C03578=1018.993,103.804,-130.711,-24.325,21.430,-41.754
C03579=1018.988,104.203,-130.749,-24.326,21.429,-41.751
C03580=1018.984,104.602,-130.786,-24.326,21.429,-41.747
C03581=1018.979,105.001,-130.824,-24.327,21.429,-41.743
C03582=1018.975,105.399,-130.861,-24.327,21.429,-41.740
C03583=1018.971,105.798,-130.899,-24.328,21.428,-41.736
C03584=1018.966,106.196,-130.936,-24.328,21.428,-41.734
C03585=1018.961,106.595,-130.974,-24.328,21.427,-41.730
C03586=1018.957,106.994,-131.011,-24.329,21.427,-41.727
C03587=1018.952,107.393,-131.049,-24.330,21.427,-41.723
C03588=1018.949,107.791,-131.087,-24.330,21.427,-41.719
C03589=1018.943,108.189,-131.124,-24.330,21.426,-41.717
C03590=1018.939,108.588,-131.162,-24.331,21.426,-41.714
C03591=1018.935,108.987,-131.199,-24.331,21.426,-41.710
C03592=1018.930,109.386,-131.237,-24.332,21.426,-41.707
C03593=1018.925,109.784,-131.275,-24.332,21.426,-41.703
C03594=1018.921,110.182,-131.312,-24.333,21.425,-41.701
C03595=1018.916,110.581,-131.350,-24.333,21.425,-41.697
C03596=1018.911,110.979,-131.388,-24.334,21.425,-41.694
C03597=1018.907,111.378,-131.425,-24.334,21.425,-41.690
C03598=1018.902,111.777,-131.463,-24.334,21.424,-41.688
C03599=1018.897,112.175,-131.500,-24.335,21.423,-41.684
C03600=1018.892,112.574,-131.539,-24.335,21.424,-41.681
C03601=1018.887,112.973,-131.577,-24.336,21.423,-41.677
C03602=1018.882,113.371,-131.613,-24.336,21.423,-41.675
C03603=1018.878,113.769,-131.652,-24.337,21.423,-41.671
C03604=1018.873,114.168,-131.689,-24.337,21.422,-41.668
C03605=1018.868,114.566,-131.727,-24.338,21.423,-41.664
C03606=1018.863,114.966,-131.765,-24.338,21.422,-41.662
C03607=1018.858,115.363,-131.803,-24.339,21.422,-41.659
C03608=1018.854,115.762,-131.840,-24.339,21.422,-41.655
C03609=1018.849,116.160,-131.878,-24.340,21.422,-41.652
C03610=1018.844,116.559,-131.916,-24.340,21.421,-41.649
C03611=1018.839,116.958,-131.953,-24.340,21.420,-41.646
C03612=1018.834,117.356,-131.991,-24.341,21.421,-41.642
C03613=1018.829,117.755,-132.029,-24.341,21.420,-41.638
C03614=1018.824,118.153,-132.067,-24.342,21.420,-41.637
C03615=1018.819,118.552,-132.105,-24.342,21.420,-41.633
C03616=1018.814,118.950,-132.143,-24.343,21.420,-41.629
C03617=1018.809,119.349,-132.180,-24.343,21.420,-41.626
C03618=1018.804,119.747,-132.218,-24.343,21.419,-41.624
C03619=1018.799,120.146,-132.256,-24.344,21.419,-41.620
C03620=1018.795,120.544,-132.294,-24.345,21.419,-41.617
C03621=1018.789,120.943,-132.332,-24.345,21.418,-41.614
C03622=1018.785,121.341,-132.370,-24.345,21.418,-41.611
C03623=1018.780,121.740,-132.408,-24.346,21.418,-41.607
C03624=1018.776,122.138,-132.447,-24.346,21.417,-41.605
C03625=1018.771,122.538,-132.484,-24.347,21.418,-41.602
C03626=1018.766,122.935,-132.522,-24.347,21.417,-41.598
C03627=1018.761,123.334,-132.561,-24.348,21.418,-41.595
C03628=1018.757,123.732,-132.599,-24.348,21.416,-41.592
C03629=1018.751,124.132,-132.637,-24.348,21.417,-41.589
C03630=1018.746,124.530,-132.675,-24.349,21.416,-41.585
C03631=1018.741,124.928,-132.714,-24.349,21.416,-41.583
C03632=1018.737,125.327,-132.751,-24.350,21.416,-41.580
C03633=1018.732,125.726,-132.790,-24.350,21.416,-41.576
C03634=1018.727,126.124,-132.828,-24.350,21.415,-41.574
C03635=1018.722,126.522,-132.867,-24.351,21.415,-41.571
C03636=1018.717,126.922,-132.904,-24.351,21.415,-41.567
C03637=1018.712,127.320,-132.943,-24.352,21.415,-41.565
C03638=1018.708,127.719,-132.981,-24.352,21.414,-41.561
C03639=1018.702,128.117,-133.019,-24.353,21.415,-41.558
C03640=1018.697,128.516,-133.057,-24.353,21.414,-41.555
C03641=1018.693,128.914,-133.096,-24.354,21.414,-41.552
C03642=1018.688,129.313,-133.134,-24.354,21.413,-41.550
C03643=1018.682,129.712,-133.172,-24.354,21.413,-41.547
C03644=1018.677,130.110,-133.210,-24.355,21.413,-41.543
C03645=1018.672,130.509,-133.249,-24.355,21.413,-41.541
C03646=1018.667,130.908,-133.287,-24.356,21.413,-41.538
C03647=1018.662,131.306,-133.325,-24.356,21.413,-41.534
C03648=1018.657,131.705,-133.364,-24.356,21.412,-41.532
C03649=1018.652,132.104,-133.402,-24.357,21.412,-41.528
C03650=1018.646,132.502,-133.440,-24.357,21.412,-41.525
C03651=1018.642,132.901,-133.479,-24.358,21.411,-41.523
C03652=1018.636,133.300,-133.517,-24.358,21.412,-41.519
C03653=1018.632,133.698,-133.555,-24.358,21.411,-41.517
C03654=1018.626,134.097,-133.594,-24.359,21.411,-41.514
C03655=1018.621,134.496,-133.632,-24.359,21.411,-41.510
C03656=1018.616,134.895,-133.671,-24.360,21.410,-41.508
C03657=1018.610,135.293,-133.710,-24.360,21.411,-41.505
C03658=1018.605,135.689,-133.747,-24.360,21.410,-41.502
C03659=1018.601,136.061,-133.783,-24.361,21.409,-41.500
C03660=1018.595,136.399,-133.815,-24.361,21.410,-41.497
C03661=1018.591,136.717,-133.846,-24.361,21.409,-41.495
C03662=1018.587,137.034,-133.876,-24.362,21.409,-41.491
C03663=1018.583,137.370,-133.909,-24.363,21.410,-41.488
C03664=1018.578,137.740,-133.944,-24.363,21.408,-41.486
C03665=1018.573,138.142,-133.983,-24.363,21.408,-41.484
C03666=1018.570,138.348,-134.003,-24.363,21.408,-41.482
C03667=1018.567,138.564,-134.024,-24.364,21.408,-41.480
C03668=1018.564,138.802,-134.047,-24.364,21.408,-41.478
C03669=1018.561,139.061,-134.072,-24.364,21.407,-41.476
C03670=1018.556,139.339,-134.099,-24.364,21.408,-41.475
C03671=1018.553,139.627,-134.126,-24.365,21.408,-41.473
C03672=1018.549,139.914,-134.154,-24.365,21.408,-41.471
C03673=1018.545,140.192,-134.182,-24.365,21.408,-41.470
C03674=1018.541,140.450,-134.206,-24.366,21.408,-41.468
C03675=1018.538,140.685,-134.229,-24.366,21.408,-41.466
C03676=1018.533,141.103,-134.269,-24.366,21.407,-41.462
C03677=1018.527,141.508,-134.308,-24.366,21.406,-41.460
C03678=1018.521,141.913,-134.347,-24.367,21.407,-41.457
C03679=1018.515,142.319,-134.386,-24.368,21.406,-41.453
C03680=1018.510,142.727,-134.425,-24.368,21.406,-41.451
C03681=1018.504,143.135,-134.466,-24.368,21.406,-41.448
C03682=1018.499,143.544,-134.505,-24.369,21.405,-41.445
C03683=1018.492,143.953,-134.544,-24.369,21.406,-41.442
C03684=1018.487,144.363,-134.584,-24.370,21.405,-41.438
C03685=1018.481,144.775,-134.624,-24.370,21.405,-41.436
C03686=1018.475,145.186,-134.664,-24.370,21.405,-41.432
C03687=1018.469,145.598,-134.704,-24.371,21.404,-41.431
C03688=1018.464,146.010,-134.743,-24.371,21.405,-41.427
C03689=1018.458,146.423,-134.783,-24.372,21.404,-41.424
C03690=1018.452,146.836,-134.823,-24.372,21.404,-41.422
C03691=1018.446,147.250,-134.863,-24.372,21.404,-41.418
C03692=1018.440,147.664,-134.904,-24.373,21.403,-41.416
C03693=1018.435,148.077,-134.943,-24.373,21.403,-41.412
C03694=1018.429,148.491,-134.983,-24.374,21.403,-41.409
C03695=1018.423,148.906,-135.023,-24.374,21.403,-41.407
C03696=1018.417,149.320,-135.064,-24.375,21.403,-41.403
C03697=1018.411,149.733,-135.103,-24.375,21.402,-41.401
C03698=1018.404,150.148,-135.144,-24.375,21.402,-41.398
C03699=1018.398,150.562,-135.184,-24.376,21.402,-41.394
C03700=1018.392,150.976,-135.224,-24.376,21.401,-41.392
C03701=1018.387,151.389,-135.264,-24.377,21.402,-41.389
C03702=1018.380,151.802,-135.304,-24.377,21.402,-41.387
C03703=1018.374,152.215,-135.345,-24.377,21.401,-41.383
C03704=1018.368,152.628,-135.384,-24.378,21.401,-41.381
C03705=1018.362,153.041,-135.424,-24.378,21.400,-41.377
C03706=1018.356,153.453,-135.465,-24.378,21.400,-41.375
C03707=1018.349,153.864,-135.504,-24.379,21.401,-41.372
C03708=1018.343,154.275,-135.544,-24.380,21.400,-41.368
C03709=1018.338,154.684,-135.584,-24.380,21.400,-41.366
C03710=1018.331,155.093,-135.624,-24.380,21.400,-41.363
C03711=1018.325,155.502,-135.663,-24.381,21.399,-41.361
C03712=1018.319,155.910,-135.703,-24.381,21.400,-41.358
C03713=1018.313,156.316,-135.742,-24.381,21.399,-41.355
C03714=1018.307,156.722,-135.782,-24.382,21.399,-41.352
C03715=1018.301,157.127,-135.821,-24.382,21.399,-41.350
C03716=1018.294,157.532,-135.861,-24.383,21.398,-41.346
C03717=1018.288,157.935,-135.899,-24.383,21.398,-41.344
C03718=1018.282,158.338,-135.939,-24.383,21.399,-41.341
C03719=1018.275,158.739,-135.978,-24.384,21.397,-41.339
C03720=1018.270,159.141,-136.017,-24.384,21.398,-41.335
C03721=1018.263,159.542,-136.055,-24.384,21.398,-41.333
C03722=1018.261,159.941,-136.098,-24.385,21.397,-41.330
C03723=1018.260,160.339,-136.139,-24.385,21.397,-41.328
C03724=1018.259,160.743,-136.182,-24.386,21.397,-41.325
C03725=1018.258,160.958,-136.203,-24.386,21.397,-41.324
C03726=1018.257,161.182,-136.227,-24.386,21.396,-41.322
C03727=1018.256,161.419,-136.252,-24.386,21.396,-41.320
C03728=1018.255,161.670,-136.279,-24.387,21.397,-41.319
C03729=1018.255,161.933,-136.307,-24.387,21.397,-41.317
C03730=1018.254,162.202,-136.334,-24.387,21.396,-41.315
C03731=1018.253,162.473,-136.362,-24.387,21.396,-41.313
C03732=1018.252,162.742,-136.392,-24.388,21.396,-41.311
C03733=1018.251,163.005,-136.419,-24.388,21.396,-41.309
C03734=1018.250,163.259,-136.445,-24.388,21.395,-41.308
C03735=1018.249,163.494,-136.470,-24.388,21.396,-41.306
C03736=1018.248,163.906,-136.513,-24.389,21.395,-41.304
C03737=1018.247,164.096,-136.533,-24.389,21.395,-41.302
C03738=1018.246,164.482,-136.574,-24.389,21.395,-41.300
C03739=1018.245,164.883,-136.616,-24.390,21.395,-41.297
C03740=1018.243,165.282,-136.658,-24.390,21.395,-41.295
C03741=1018.242,165.683,-136.700,-24.390,21.394,-41.291
C03742=1018.241,166.084,-136.743,-24.391,21.394,-41.289
C03743=1018.239,166.483,-136.785,-24.391,21.395,-41.286
C03744=1018.238,166.884,-136.827,-24.391,21.393,-41.284
C03745=1018.237,167.285,-136.870,-24.392,21.394,-41.280
C03746=1018.235,167.685,-136.911,-24.392,21.394,-41.278
C03747=1018.234,168.085,-136.954,-24.393,21.394,-41.275
C03748=1018.233,168.486,-136.996,-24.393,21.393,-41.273
C03749=1018.232,168.887,-137.039,-24.393,21.393,-41.271
C03750=1018.231,169.287,-137.081,-24.394,21.393,-41.267
C03751=1018.229,169.687,-137.123,-24.394,21.392,-41.265
C03752=1018.228,170.087,-137.165,-24.395,21.392,-41.262
C03753=1018.227,170.489,-137.208,-24.395,21.392,-41.260
C03754=1018.225,170.889,-137.250,-24.395,21.392,-41.256
C03755=1018.225,171.289,-137.293,-24.396,21.392,-41.254
C03756=1018.223,171.690,-137.335,-24.396,21.392,-41.251
C03757=1018.222,172.091,-137.378,-24.396,21.392,-41.249
C03758=1018.221,172.491,-137.420,-24.397,21.391,-41.247
C03759=1018.219,172.892,-137.463,-24.397,21.391,-41.243
C03760=1018.218,173.293,-137.506,-24.397,21.391,-41.242
C03761=1018.217,173.693,-137.548,-24.398,21.390,-41.238
C03762=1018.216,174.094,-137.590,-24.398,21.390,-41.236
C03763=1018.214,174.495,-137.633,-24.399,21.391,-41.233
C03764=1018.213,174.895,-137.676,-24.399,21.390,-41.231
C03765=1018.212,175.296,-137.718,-24.400,21.390,-41.227
C03766=1018.211,175.697,-137.761,-24.400,21.390,-41.225
C03767=1018.210,176.098,-137.804,-24.400,21.390,-41.223
C03768=1018.209,176.498,-137.847,-24.401,21.389,-41.219
C03769=1018.207,176.899,-137.889,-24.401,21.389,-41.218
C03770=1018.206,177.299,-137.931,-24.401,21.389,-41.214
C03771=1018.206,177.701,-137.975,-24.402,21.389,-41.212
C03772=1018.204,178.101,-138.018,-24.402,21.389,-41.209
C03773=1018.203,178.502,-138.060,-24.402,21.388,-41.207
C03774=1018.202,178.904,-138.103,-24.403,21.388,-41.205
C03775=1018.201,179.304,-138.146,-24.403,21.388,-41.201
C03776=1018.200,179.704,-138.189,-24.403,21.388,-41.199
C03777=1018.199,180.105,-138.232,-24.404,21.388,-41.196
C03778=1018.198,180.506,-138.275,-24.404,21.388,-41.194
C03779=1018.197,180.908,-138.317,-24.405,21.387,-41.190
C03780=1018.195,181.308,-138.360,-24.405,21.387,-41.188
C03781=1018.194,181.709,-138.403,-24.405,21.387,-41.186
C03782=1018.193,182.110,-138.447,-24.406,21.387,-41.183
C03783=1018.192,182.511,-138.490,-24.406,21.386,-41.181
C03784=1018.191,182.912,-138.533,-24.407,21.387,-41.177
C03785=1018.190,183.312,-138.576,-24.407,21.386,-41.176
C03786=1018.189,183.713,-138.619,-24.407,21.386,-41.172
C03787=1018.188,184.115,-138.662,-24.408,21.386,-41.170
C03788=1018.187,184.515,-138.705,-24.408,21.386,-41.168
C03789=1018.186,184.917,-138.748,-24.409,21.386,-41.165
C03790=1018.185,185.318,-138.791,-24.409,21.385,-41.162
C03791=1018.184,185.719,-138.834,-24.409,21.385,-41.159
C03792=1018.183,186.120,-138.878,-24.410,21.385,-41.157
C03793=1018.182,186.521,-138.921,-24.410,21.384,-41.155
C03794=1018.181,186.922,-138.964,-24.410,21.384,-41.151
C03795=1018.180,187.323,-139.007,-24.411,21.384,-41.150
C03796=1018.180,187.723,-139.051,-24.411,21.385,-41.146
C03797=1018.179,188.125,-139.095,-24.411,21.384,-41.144
C03798=1018.178,188.525,-139.137,-24.412,21.384,-41.141
C03799=1018.177,188.926,-139.181,-24.412,21.384,-41.139
C03800=1018.176,189.328,-139.224,-24.412,21.384,-41.137
C03801=1018.176,189.729,-139.267,-24.413,21.383,-41.133
C03802=1018.175,190.130,-139.311,-24.413,21.383,-41.131
C03803=1018.174,190.531,-139.354,-24.414,21.383,-41.128
C03804=1018.173,190.932,-139.397,-24.414,21.383,-41.126
C03805=1018.172,191.333,-139.442,-24.414,21.382,-41.124
C03806=1018.171,191.734,-139.485,-24.415,21.382,-41.120
C03807=1018.170,192.135,-139.528,-24.415,21.382,-41.118
C03808=1018.169,192.536,-139.572,-24.415,21.382,-41.115
C03809=1018.169,192.938,-139.615,-24.416,21.382,-41.113
C03810=1018.168,193.338,-139.659,-24.416,21.382,-41.109
C03811=1018.167,193.739,-139.702,-24.417,21.382,-41.108
C03812=1018.166,194.141,-139.746,-24.417,21.381,-41.105
C03813=1018.165,194.541,-139.790,-24.417,21.381,-41.102
C03814=1018.165,194.943,-139.833,-24.418,21.381,-41.100
C03815=1018.164,195.345,-139.877,-24.418,21.381,-41.097
C03816=1018.164,195.745,-139.921,-24.418,21.380,-41.094
C03817=1018.163,196.147,-139.965,-24.419,21.381,-41.091
C03818=1018.162,196.548,-140.008,-24.419,21.380,-41.089
C03819=1018.161,196.949,-140.052,-24.419,21.380,-41.087
C03820=1018.161,197.350,-140.096,-24.420,21.380,-41.084
C03821=1018.160,197.750,-140.140,-24.420,21.380,-41.082
C03822=1018.159,198.153,-140.184,-24.421,21.380,-41.078
C03823=1018.159,198.554,-140.227,-24.421,21.379,-41.076
C03824=1018.158,198.954,-140.271,-24.421,21.379,-41.074
C03825=1018.158,199.353,-140.315,-24.422,21.379,-41.071
C03826=1018.157,199.742,-140.358,-24.422,21.379,-41.069
C03827=1018.156,200.142,-140.401,-24.423,21.378,-41.065
C03828=1018.156,200.355,-140.425,-24.423,21.378,-41.065
C03829=1018.156,200.577,-140.449,-24.423,21.378,-41.063
C03830=1018.156,200.807,-140.475,-24.423,21.378,-41.061
C03831=1018.155,201.034,-140.500,-24.423,21.379,-41.060
C03832=1018.154,201.442,-140.544,-24.424,21.378,-41.058
C03833=1018.154,201.793,-140.582,-24.424,21.378,-41.054
C03834=1018.155,202.143,-140.622,-24.424,21.378,-41.052
C03835=1018.156,202.530,-140.666,-24.425,21.378,-41.051
C03836=1018.162,203.746,-140.801,-24.373,21.403,-41.416
C03837=1018.164,203.994,-140.828,-24.373,21.404,-41.415
C03838=1018.166,204.242,-140.857,-24.373,21.403,-41.414
C03839=1018.168,204.491,-140.884,-24.373,21.403,-41.412
C03840=1018.170,204.739,-140.911,-24.374,21.404,-41.411
C03841=1018.172,204.988,-140.939,-24.373,21.403,-41.410
C03842=1018.174,205.237,-140.966,-24.374,21.403,-41.409
C03843=1018.176,205.486,-140.994,-24.374,21.403,-41.407
C03844=1018.178,205.734,-141.021,-24.374,21.402,-41.407
C03845=1018.180,205.982,-141.049,-24.374,21.403,-41.405
C03846=1018.181,206.231,-141.076,-24.375,21.403,-41.403
C03847=1018.184,206.479,-141.104,-24.375,21.402,-41.401
C03848=1018.186,206.727,-141.131,-24.375,21.402,-41.401
C03849=1018.187,206.976,-141.158,-24.375,21.402,-41.399
C03850=1018.189,207.224,-141.186,-24.375,21.402,-41.398
C03851=1018.192,207.473,-141.213,-24.375,21.402,-41.398
C03852=1018.193,207.722,-141.241,-24.376,21.402,-41.396
C03853=1018.196,207.970,-141.269,-24.376,21.402,-41.394
C03854=1018.198,208.218,-141.296,-24.376,21.402,-41.392
C03855=1018.199,208.461,-141.323,-24.376,21.401,-41.392
C03856=1018.201,208.704,-141.350,-24.376,21.402,-41.391
C03857=1018.203,208.946,-141.377,-24.377,21.402,-41.389
C03858=1018.206,209.189,-141.404,-24.377,21.401,-41.388
C03859=1018.208,209.432,-141.430,-24.377,21.402,-41.387
C03860=1018.209,209.675,-141.458,-24.377,21.401,-41.385
C03861=1018.212,209.917,-141.485,-24.377,21.401,-41.383
C03862=1018.213,210.160,-141.512,-24.377,21.401,-41.383
C03863=1018.216,210.408,-141.540,-24.378,21.401,-41.381
C03864=1018.217,210.657,-141.567,-24.378,21.401,-41.379
C03865=1018.220,210.905,-141.595,-24.378,21.401,-41.378
C03866=1018.222,211.153,-141.622,-24.378,21.400,-41.377
C03867=1018.224,211.402,-141.651,-24.378,21.400,-41.375
C03868=1018.226,211.651,-141.677,-24.379,21.401,-41.374
C03869=1018.228,211.899,-141.706,-24.379,21.401,-41.372
C03870=1018.230,212.148,-141.733,-24.379,21.400,-41.372
C03871=1018.233,212.396,-141.761,-24.379,21.400,-41.370
C03872=1018.234,212.644,-141.789,-24.380,21.400,-41.368
C03873=1018.236,212.893,-141.816,-24.380,21.400,-41.366
C03874=1018.239,213.141,-141.844,-24.380,21.400,-41.366
C03875=1018.241,213.460,-141.879,-24.380,21.400,-41.365
C03876=1018.244,213.778,-141.915,-24.380,21.400,-41.363
C03877=1018.247,214.097,-141.951,-24.381,21.399,-41.361
C03878=1018.250,214.416,-141.986,-24.381,21.399,-41.359
C03879=1018.252,214.665,-142.015,-24.381,21.399,-41.357
C03880=1018.254,214.912,-142.042,-24.381,21.400,-41.356
C03881=1018.256,215.160,-142.070,-24.382,21.399,-41.354
C03882=1018.258,215.410,-142.098,-24.382,21.399,-41.352
C03883=1018.262,215.825,-142.145,-24.382,21.399,-41.350
C03884=1018.266,216.240,-142.191,-24.382,21.399,-41.348
C03885=1018.270,216.656,-142.237,-24.383,21.399,-41.345
C03886=1018.274,217.071,-142.284,-24.383,21.398,-41.342
C03887=1018.276,217.319,-142.311,-24.383,21.399,-41.341
C03888=1018.278,217.568,-142.340,-24.384,21.398,-41.339
C03889=1018.281,217.816,-142.368,-24.384,21.397,-41.339
C03890=1018.282,218.065,-142.395,-24.384,21.397,-41.337
C03891=1018.285,218.314,-142.423,-24.384,21.398,-41.335
C03892=1018.287,218.561,-142.451,-24.384,21.398,-41.333
C03893=1018.289,218.810,-142.480,-24.385,21.397,-41.332
C03894=1018.292,219.058,-142.508,-24.385,21.397,-41.330
C03895=1018.294,219.307,-142.535,-24.385,21.397,-41.330
C03896=1018.296,219.556,-142.563,-24.385,21.397,-41.328
C03897=1018.298,219.804,-142.591,-24.385,21.397,-41.326
C03898=1018.301,220.052,-142.619,-24.386,21.397,-41.324
C03899=1018.303,220.300,-142.647,-24.386,21.397,-41.323
C03900=1018.306,220.549,-142.675,-24.386,21.397,-41.321
C03901=1018.308,220.797,-142.703,-24.386,21.396,-41.320
C03902=1018.311,221.046,-142.732,-24.386,21.396,-41.318
C03903=1018.313,221.294,-142.759,-24.387,21.397,-41.317
C03904=1018.316,221.542,-142.787,-24.387,21.396,-41.315
C03905=1018.318,221.791,-142.816,-24.387,21.396,-41.313
C03906=1018.320,222.040,-142.843,-24.388,21.396,-41.311
C03907=1018.322,222.282,-142.870,-24.388,21.397,-41.310
C03908=1018.325,222.526,-142.898,-24.388,21.396,-41.309
C03909=1018.327,222.768,-142.926,-24.388,21.395,-41.308
C03910=1018.330,223.011,-142.953,-24.388,21.395,-41.306
C03911=1018.332,223.254,-142.981,-24.389,21.396,-41.304
C03912=1018.334,223.497,-143.008,-24.389,21.396,-41.302
C03913=1018.337,223.740,-143.036,-24.389,21.395,-41.300
C03914=1018.339,223.983,-143.063,-24.389,21.395,-41.300
C03915=1018.342,224.231,-143.092,-24.389,21.394,-41.298
C03916=1018.344,224.479,-143.119,-24.390,21.395,-41.297
C03917=1018.346,224.728,-143.148,-24.390,21.395,-41.295
C03918=1018.349,224.976,-143.177,-24.390,21.395,-41.293
C03919=1018.352,225.224,-143.204,-24.390,21.394,-41.291
C03920=1018.354,225.473,-143.233,-24.391,21.394,-41.289
C03921=1018.356,225.721,-143.261,-24.391,21.395,-41.288
C03922=1018.359,225.969,-143.289,-24.391,21.395,-41.286
C03923=1018.361,226.218,-143.317,-24.391,21.394,-41.285
C03924=1018.364,226.466,-143.345,-24.391,21.393,-41.284
C03925=1018.366,226.715,-143.374,-24.392,21.393,-41.282
C03926=1018.369,226.964,-143.402,-24.392,21.394,-41.280
C03927=1018.372,227.211,-143.430,-24.392,21.394,-41.278
C03928=1018.374,227.460,-143.459,-24.393,21.393,-41.276
C03929=1018.377,227.709,-143.487,-24.393,21.393,-41.275
C03930=1018.379,227.956,-143.515,-24.393,21.393,-41.273
C03931=1018.381,228.205,-143.543,-24.393,21.394,-41.271
C03932=1018.384,228.454,-143.571,-24.394,21.393,-41.269
C03933=1018.388,228.702,-143.600,-24.394,21.393,-41.267
C03934=1018.389,228.950,-143.629,-24.394,21.393,-41.266
C03935=1018.392,229.193,-143.656,-24.394,21.392,-41.265
C03936=1018.395,229.437,-143.684,-24.394,21.392,-41.263
C03937=1018.397,229.679,-143.711,-24.395,21.392,-41.262
C03938=1018.400,229.922,-143.740,-24.395,21.392,-41.260
C03939=1018.403,230.165,-143.767,-24.395,21.392,-41.258
C03940=1018.405,230.408,-143.795,-24.395,21.392,-41.256
C03941=1018.408,230.651,-143.823,-24.396,21.392,-41.254
C03942=1018.410,230.895,-143.851,-24.396,21.391,-41.252
C03943=1018.413,231.143,-143.880,-24.396,21.392,-41.251
C03944=1018.416,231.391,-143.907,-24.396,21.392,-41.249
C03945=1018.418,231.640,-143.936,-24.397,21.392,-41.247
C03946=1018.421,231.888,-143.965,-24.397,21.391,-41.245
C03947=1018.424,232.136,-143.993,-24.397,21.391,-41.243
C03948=1018.426,232.384,-144.022,-24.397,21.391,-41.242
C03949=1018.429,232.633,-144.050,-24.398,21.391,-41.240
C03950=1018.432,232.881,-144.078,-24.398,21.390,-41.238
C03951=1018.434,233.129,-144.107,-24.398,21.391,-41.236
C03952=1018.437,233.378,-144.135,-24.399,21.391,-41.234
C03953=1018.440,233.626,-144.165,-24.399,21.391,-41.233
C03954=1018.443,233.875,-144.193,-24.399,21.390,-41.231
C03955=1018.446,234.123,-144.221,-24.399,21.390,-41.229
C03956=1018.448,234.372,-144.250,-24.400,21.390,-41.227
C03957=1018.451,234.620,-144.278,-24.400,21.390,-41.225
C03958=1018.453,234.868,-144.307,-24.400,21.390,-41.223
C03959=1018.456,235.116,-144.335,-24.400,21.389,-41.221
C03960=1018.459,235.364,-144.364,-24.401,21.389,-41.219
C03961=1018.462,235.613,-144.393,-24.401,21.389,-41.218
C03962=1018.465,235.861,-144.422,-24.401,21.390,-41.216
C03963=1018.468,236.104,-144.449,-24.401,21.389,-41.214
C03964=1018.470,236.347,-144.478,-24.402,21.389,-41.212
C03965=1018.473,236.590,-144.506,-24.402,21.389,-41.210
C03966=1018.476,236.834,-144.534,-24.402,21.389,-41.209
C03967=1018.479,237.077,-144.562,-24.402,21.388,-41.207
C03968=1018.481,237.320,-144.590,-24.403,21.388,-41.205
C03969=1018.484,237.563,-144.618,-24.403,21.388,-41.203
C03970=1018.487,237.806,-144.646,-24.403,21.388,-41.201
C03971=1018.490,238.054,-144.675,-24.403,21.388,-41.199
C03972=1018.493,238.303,-144.703,-24.404,21.387,-41.197
C03973=1018.495,238.551,-144.733,-24.404,21.387,-41.195
C03974=1018.499,238.799,-144.762,-24.405,21.388,-41.192
C03975=1018.501,239.048,-144.790,-24.405,21.387,-41.190
C03976=1018.504,239.296,-144.819,-24.405,21.387,-41.188
C03977=1018.507,239.544,-144.848,-24.405,21.387,-41.186
C03978=1018.510,239.793,-144.876,-24.406,21.387,-41.184
C03979=1018.513,240.041,-144.905,-24.406,21.386,-41.183
C03980=1018.517,240.290,-144.934,-24.406,21.386,-41.181
C03981=1018.519,240.538,-144.964,-24.406,21.386,-41.179
C03982=1018.522,240.786,-144.992,-24.407,21.386,-41.177
C03983=1018.525,241.034,-145.021,-24.407,21.386,-41.174
C03984=1018.528,241.283,-145.050,-24.407,21.386,-41.172
C03985=1018.531,241.531,-145.079,-24.408,21.386,-41.170
C03986=1018.533,241.780,-145.107,-24.408,21.386,-41.168
C03987=1018.537,242.028,-145.136,-24.408,21.385,-41.166
C03988=1018.540,242.275,-145.165,-24.408,21.385,-41.164
C03989=1018.543,242.524,-145.195,-24.409,21.385,-41.162
C03990=1018.546,242.772,-145.224,-24.409,21.385,-41.159
C03991=1018.549,243.016,-145.252,-24.410,21.385,-41.157
C03992=1018.552,243.259,-145.280,-24.410,21.385,-41.155
C03993=1018.555,243.502,-145.309,-24.410,21.385,-41.153
C03994=1018.558,243.745,-145.337,-24.410,21.384,-41.151
C03995=1018.560,243.988,-145.366,-24.411,21.384,-41.150
C03996=1018.564,244.232,-145.394,-24.411,21.384,-41.148
C03997=1018.567,244.475,-145.422,-24.411,21.384,-41.144
C03998=1018.570,244.718,-145.451,-24.412,21.384,-41.143
C03999=1018.573,244.967,-145.480,-24.412,21.384,-41.141
C04000=1018.576,245.215,-145.509,-24.412,21.384,-41.139
C04001=1018.579,245.463,-145.538,-24.412,21.384,-41.137
C04002=1018.582,245.711,-145.567,-24.413,21.384,-41.134
C04003=1018.586,245.960,-145.596,-24.413,21.384,-41.132
C04004=1018.588,246.208,-145.626,-24.413,21.383,-41.129
C04005=1018.592,246.456,-145.655,-24.414,21.382,-41.127
C04006=1018.595,246.704,-145.683,-24.414,21.382,-41.126
C04007=1018.598,246.953,-145.713,-24.414,21.383,-41.122
C04008=1018.601,247.201,-145.742,-24.415,21.382,-41.120
C04009=1018.604,247.449,-145.771,-24.415,21.382,-41.118
C04010=1018.607,247.697,-145.800,-24.415,21.382,-41.117
C04011=1018.610,247.946,-145.830,-24.416,21.382,-41.113
C04012=1018.613,248.194,-145.859,-24.416,21.382,-41.111
C04013=1018.617,248.443,-145.888,-24.416,21.381,-41.109
C04014=1018.620,248.690,-145.918,-24.417,21.381,-41.107
C04015=1018.623,248.938,-145.947,-24.417,21.381,-41.104
C04016=1018.627,249.187,-145.976,-24.417,21.381,-41.102
C04017=1018.630,249.435,-146.005,-24.418,21.381,-41.100
C04018=1018.632,249.684,-146.035,-24.418,21.381,-41.098
C04019=1018.636,249.927,-146.063,-24.418,21.381,-41.095
C04020=1018.639,250.171,-146.092,-24.419,21.381,-41.093
C04021=1018.643,250.413,-146.121,-24.419,21.380,-41.091
C04022=1018.646,250.657,-146.150,-24.419,21.380,-41.089
C04023=1018.649,250.901,-146.178,-24.420,21.380,-41.085
C04024=1018.652,251.144,-146.207,-24.420,21.380,-41.084
C04025=1018.655,251.387,-146.236,-24.420,21.380,-41.082
C04026=1018.659,251.631,-146.265,-24.421,21.380,-41.078
C04027=1018.661,251.879,-146.294,-24.421,21.380,-41.076
C04028=1018.666,252.127,-146.324,-24.421,21.379,-41.074
C04029=1018.668,252.375,-146.353,-24.421,21.378,-41.072
C04030=1018.671,252.623,-146.382,-24.422,21.379,-41.069
C04031=1018.675,252.872,-146.412,-24.422,21.379,-41.067
C04032=1018.678,253.120,-146.441,-24.423,21.378,-41.065
C04033=1018.681,253.369,-146.471,-24.423,21.378,-41.061
C04034=1018.685,253.616,-146.500,-24.423,21.378,-41.060
C04035=1018.689,253.865,-146.530,-24.424,21.378,-41.058
C04036=1018.691,254.112,-146.560,-24.424,21.378,-41.054
C04037=1018.695,254.361,-146.589,-24.424,21.378,-41.052
C04038=1018.698,254.609,-146.618,-24.425,21.377,-41.049
C04039=1018.702,254.857,-146.648,-24.425,21.377,-41.047
C04040=1018.705,255.106,-146.678,-24.425,21.377,-41.045
C04041=1018.709,255.354,-146.707,-24.426,21.377,-41.042
C04042=1018.712,255.603,-146.737,-24.426,21.377,-41.040
C04043=1018.715,255.850,-146.767,-24.426,21.376,-41.037
C04044=1018.718,256.099,-146.796,-24.427,21.376,-41.034
C04045=1018.723,256.347,-146.826,-24.427,21.376,-41.032
C04046=1018.725,256.595,-146.856,-24.428,21.377,-41.029
C04047=1018.729,256.839,-146.884,-24.428,21.376,-41.027
C04048=1018.732,257.082,-146.913,-24.428,21.375,-41.025
C04049=1018.735,257.326,-146.943,-24.429,21.376,-41.021
C04050=1018.739,257.568,-146.972,-24.429,21.376,-41.019
C04051=1018.743,257.812,-147.001,-24.429,21.375,-41.018
C04052=1018.746,258.056,-147.030,-24.430,21.375,-41.014
C04053=1018.750,258.299,-147.059,-24.430,21.375,-41.012
C04054=1018.767,259.535,-147.213,-24.551,21.322,-40.171
C04055=1018.770,259.815,-147.250,-24.587,21.310,-39.930
C04056=1018.772,260.095,-147.287,-24.622,21.298,-39.688
C04057=1018.774,260.374,-147.326,-24.658,21.287,-39.446
C04058=1018.775,260.654,-147.364,-24.693,21.275,-39.204
C04059=1018.776,260.901,-147.398,-24.725,21.267,-38.988
C04060=1018.776,261.149,-147.433,-24.758,21.259,-38.770
C04061=1018.776,261.396,-147.469,-24.790,21.251,-38.554
C04062=1018.776,261.644,-147.505,-24.823,21.245,-38.337
C04063=1018.776,261.924,-147.546,-24.860,21.238,-38.090
C04064=1018.775,262.203,-147.589,-24.897,21.233,-37.842
C04065=1018.773,262.482,-147.632,-24.935,21.227,-37.593
C04066=1018.770,262.761,-147.675,-24.973,21.223,-37.345
C04067=1018.769,263.008,-147.713,-25.006,21.220,-37.124
C04068=1018.767,263.255,-147.753,-25.040,21.217,-36.903
C04069=1018.764,263.502,-147.793,-25.074,21.216,-36.681
C04070=1018.760,263.749,-147.833,-25.108,21.215,-36.458
C04071=1018.755,264.028,-147.880,-25.147,21.216,-36.205
C04072=1018.752,264.307,-147.928,-25.186,21.217,-35.952
C04073=1018.747,264.586,-147.975,-25.226,21.219,-35.699
C04074=1018.741,264.865,-148.023,-25.265,21.221,-35.444
C04075=1018.736,265.112,-148.067,-25.300,21.225,-35.219
C04076=1018.730,265.358,-148.111,-25.335,21.229,-34.991
C04077=1018.724,265.604,-148.154,-25.370,21.233,-34.766
C04078=1018.718,265.850,-148.199,-25.406,21.239,-34.538
C04079=1018.710,266.128,-148.251,-25.446,21.246,-34.279
C04080=1018.702,266.408,-148.303,-25.487,21.254,-34.021
C04081=1018.693,266.686,-148.356,-25.527,21.264,-33.760
C04082=1018.684,266.965,-148.409,-25.568,21.275,-33.499
C04083=1018.677,267.210,-148.457,-25.604,21.284,-33.269
C04084=1018.667,267.455,-148.505,-25.641,21.295,-33.037
C04085=1018.658,267.701,-148.554,-25.677,21.306,-32.805
C04086=1018.649,267.946,-148.604,-25.714,21.319,-32.571
C04087=1018.638,268.224,-148.659,-25.755,21.333,-32.307
C04088=1018.627,268.503,-148.717,-25.797,21.350,-32.039
C04089=1018.614,268.782,-148.775,-25.839,21.367,-31.772
C04090=1018.601,269.060,-148.833,-25.881,21.386,-31.502
C04091=1018.590,269.304,-148.885,-25.918,21.402,-31.266
C04092=1018.578,269.549,-148.937,-25.955,21.420,-31.029
C04093=1018.566,269.792,-148.991,-25.992,21.439,-30.791
C04094=1018.554,270.037,-149.045,-26.030,21.459,-30.551
C04095=1018.539,270.315,-149.107,-26.072,21.483,-30.277
C04096=1018.524,270.594,-149.169,-26.115,21.507,-30.003
C04097=1018.508,270.871,-149.232,-26.158,21.533,-29.728
C04098=1018.491,271.150,-149.296,-26.201,21.560,-29.450
C04099=1018.477,271.393,-149.352,-26.238,21.585,-29.208
C04100=1018.462,271.636,-149.409,-26.276,21.610,-28.964
C04101=1018.447,271.879,-149.467,-26.314,21.637,-28.720
C04102=1018.432,272.122,-149.524,-26.351,21.664,-28.476
C04103=1018.413,272.400,-149.592,-26.395,21.697,-28.194
C04104=1018.393,272.678,-149.659,-26.438,21.731,-27.910
C04105=1018.374,272.957,-149.728,-26.481,21.766,-27.626
C04106=1018.354,273.234,-149.796,-26.525,21.803,-27.342
C04107=1018.337,273.476,-149.858,-26.562,21.835,-27.092
C04108=1018.318,273.717,-149.918,-26.600,21.869,-26.841
C04109=1018.300,273.959,-149.981,-26.638,21.903,-26.590
C04110=1018.281,274.201,-150.042,-26.676,21.940,-26.336
C04111=1018.259,274.478,-150.115,-26.720,21.983,-26.043
C04112=1018.236,274.756,-150.188,-26.763,22.027,-25.750
C04113=1018.213,275.034,-150.262,-26.807,22.073,-25.453
C04114=1018.190,275.311,-150.337,-26.851,22.119,-25.156
C04115=1018.169,275.551,-150.402,-26.889,22.162,-24.896
C04116=1018.147,275.792,-150.467,-26.927,22.204,-24.635
C04117=1018.125,276.033,-150.534,-26.965,22.250,-24.373
C04118=1018.104,276.272,-150.601,-27.003,22.295,-24.109
C04119=1018.077,276.549,-150.679,-27.046,22.349,-23.804
C04120=1018.051,276.827,-150.758,-27.090,22.404,-23.496
C04121=1018.024,277.104,-150.837,-27.134,22.462,-23.186
C04122=1017.996,277.381,-150.917,-27.177,22.521,-22.877
C04123=1017.972,277.620,-150.987,-27.215,22.573,-22.606
C04124=1017.948,277.859,-151.057,-27.252,22.626,-22.334
C04125=1017.922,278.097,-151.128,-27.290,22.681,-22.062
C04126=1017.896,278.335,-151.200,-27.327,22.737,-21.789
C04127=1017.867,278.612,-151.283,-27.370,22.804,-21.469
C04128=1017.836,278.889,-151.367,-27.413,22.873,-21.147
C04129=1017.805,279.165,-151.453,-27.456,22.942,-20.824
C04130=1017.774,279.442,-151.538,-27.498,23.014,-20.499
C04131=1017.746,279.679,-151.612,-27.534,23.078,-20.218
C04132=1017.718,279.916,-151.687,-27.570,23.142,-19.936
C04133=1017.689,280.153,-151.763,-27.606,23.208,-19.653
C04134=1017.661,280.389,-151.839,-27.642,23.276,-19.367
C04135=1017.626,280.666,-151.928,-27.684,23.357,-19.031
C04136=1017.592,280.941,-152.019,-27.725,23.440,-18.691
C04137=1017.557,281.217,-152.109,-27.766,23.526,-18.349
C04138=1017.522,281.493,-152.201,-27.807,23.613,-18.004
C04139=1017.490,281.728,-152.280,-27.842,23.690,-17.706
C04140=1017.459,281.963,-152.360,-27.877,23.768,-17.406
C04141=1017.427,282.198,-152.440,-27.911,23.848,-17.104
C04142=1017.395,282.433,-152.520,-27.945,23.929,-16.801
C04143=1017.356,282.708,-152.616,-27.984,24.027,-16.441
C04144=1017.318,282.983,-152.712,-28.023,24.128,-16.079
C04145=1017.278,283.258,-152.809,-28.062,24.232,-15.713
C04146=1017.237,283.532,-152.907,-28.100,24.338,-15.343
C04147=1017.203,283.765,-152.991,-28.132,24.429,-15.026
C04148=1017.169,283.998,-153.076,-28.164,24.524,-14.708
C04149=1017.133,284.231,-153.161,-28.195,24.619,-14.388
C04150=1017.097,284.463,-153.246,-28.226,24.716,-14.065
C04151=1017.054,284.737,-153.348,-28.261,24.835,-13.680
C04152=1017.010,285.011,-153.451,-28.296,24.955,-13.292
C04153=1016.966,285.285,-153.555,-28.330,25.079,-12.901
C04154=1016.922,285.558,-153.659,-28.364,25.204,-12.507
C04155=1016.883,285.789,-153.747,-28.391,25.314,-12.171
C04156=1016.845,286.019,-153.837,-28.418,25.425,-11.832
C04157=1016.806,286.250,-153.928,-28.444,25.537,-11.492
C04158=1016.767,286.479,-154.018,-28.470,25.652,-11.148
C04159=1016.719,286.752,-154.126,-28.499,25.792,-10.737
C04160=1016.670,287.025,-154.235,-28.527,25.936,-10.320
C04161=1016.622,287.297,-154.345,-28.555,26.082,-9.899
C04162=1016.572,287.569,-154.457,-28.581,26.233,-9.471
C04163=1016.530,287.796,-154.551,-28.602,26.363,-9.109
C04164=1016.488,288.024,-154.645,-28.622,26.495,-8.743
C04165=1016.445,288.252,-154.740,-28.641,26.630,-8.372
C04166=1016.401,288.478,-154.836,-28.659,26.767,-7.999
C04167=1016.349,288.750,-154.952,-28.679,26.937,-7.545
C04168=1016.296,289.021,-155.068,-28.698,27.109,-7.088
C04169=1016.241,289.292,-155.185,-28.715,27.285,-6.624
C04170=1016.188,289.561,-155.304,-28.730,27.467,-6.153
C04171=1016.141,289.786,-155.404,-28.742,27.622,-5.757
C04172=1016.095,290.011,-155.503,-28.752,27.779,-5.357
C04173=1016.048,290.235,-155.604,-28.760,27.939,-4.952
C04174=1016.000,290.459,-155.705,-28.767,28.103,-4.544
C04175=1015.942,290.728,-155.828,-28.773,28.305,-4.046
C04176=1015.884,290.997,-155.951,-28.777,28.512,-3.541
C04177=1015.825,291.265,-156.077,-28.778,28.722,-3.030
C04178=1015.765,291.534,-156.202,-28.777,28.937,-2.514
C04179=1015.715,291.755,-156.307,-28.773,29.120,-2.080
C04180=1015.664,291.976,-156.413,-28.768,29.306,-1.642
C04181=1015.613,292.196,-156.519,-28.761,29.494,-1.200
C04182=1015.561,292.417,-156.626,-28.751,29.688,-0.751
C04183=1015.498,292.683,-156.757,-28.736,29.926,-0.203
C04184=1015.434,292.950,-156.888,-28.717,30.168,0.353
C04185=1015.369,293.216,-157.022,-28.695,30.417,0.916
C04186=1015.303,293.481,-157.155,-28.669,30.673,1.490
C04187=1015.249,293.698,-157.266,-28.645,30.886,1.967
C04188=1015.194,293.915,-157.377,-28.617,31.104,2.450
C04189=1015.138,294.132,-157.490,-28.586,31.327,2.940
C04190=1015.081,294.349,-157.603,-28.552,31.552,3.436
C04191=1015.012,294.612,-157.742,-28.506,31.835,4.050
C04192=1014.943,294.875,-157.882,-28.455,32.122,4.672
C04193=1014.871,295.138,-158.023,-28.398,32.417,5.306
C04194=1014.800,295.400,-158.165,-28.335,32.716,5.947
C04195=1014.740,295.613,-158.283,-28.280,32.966,6.479
C04196=1014.681,295.826,-158.400,-28.220,33.220,7.016
C04197=1014.620,296.038,-158.518,-28.156,33.478,7.560
C04198=1014.560,296.250,-158.637,-28.087,33.740,8.111
C04199=1014.484,296.510,-158.785,-27.996,34.069,8.801
C04200=1014.408,296.770,-158.934,-27.897,34.404,9.500
C04201=1014.330,297.029,-159.084,-27.790,34.746,10.213
C04202=1014.252,297.287,-159.235,-27.675,35.094,10.935
C04203=1014.188,297.495,-159.359,-27.576,35.380,11.529
C04204=1014.124,297.703,-159.483,-27.470,35.670,12.129
C04205=1014.059,297.910,-159.607,-27.359,35.964,12.737
C04206=1013.994,298.116,-159.733,-27.241,36.263,13.354
C04207=1013.910,298.373,-159.890,-27.085,36.640,14.133
C04208=1013.827,298.628,-160.048,-26.918,37.024,14.926
C04209=1013.743,298.883,-160.208,-26.741,37.414,15.733
C04210=1013.657,299.137,-160.369,-26.551,37.810,16.553
C04211=1013.589,299.340,-160.499,-26.391,38.132,17.220
C04212=1013.520,299.541,-160.629,-26.221,38.458,17.898
C04213=1013.449,299.743,-160.760,-26.044,38.788,18.586
C04214=1013.378,299.944,-160.892,-25.857,39.121,19.283
///RCONF 0,0,0,0,0,0,0,0,0,0,0,0,0,0,0,0,0,0,0,0,0,0,0,0
C04215=1013.289,300.196,-161.059,-25.611,39.544,20.170
C04216=1013.199,300.446,-161.227,-25.349,39.974,21.077
C04217=1013.108,300.696,-161.397,-25.071,40.409,21.999
C04218=1013.014,300.945,-161.567,-24.778,40.847,22.938
C04219=1012.941,301.141,-161.703,-24.533,41.199,23.695
C04220=1012.866,301.337,-161.841,-24.278,41.553,24.463
C04221=1012.791,301.532,-161.978,-24.010,41.911,25.245
C04222=1012.716,301.727,-162.116,-23.731,42.271,26.037
C04223=1012.619,301.973,-162.293,-23.359,42.732,27.060
C04224=1012.521,302.217,-162.472,-22.967,43.196,28.105
C04225=1012.422,302.462,-162.651,-22.552,43.665,29.173
C04226=1012.322,302.704,-162.832,-22.115,44.137,30.264
C04227=1012.243,302.894,-162.974,-21.757,44.508,31.133
C04228=1012.163,303.083,-163.118,-21.384,44.880,32.017
C04229=1012.082,303.271,-163.262,-20.996,45.254,32.916
C04230=1012.002,303.459,-163.408,-20.592,45.628,33.828
C04231=1011.897,303.698,-163.595,-20.052,46.107,35.019
C04232=1011.792,303.937,-163.784,-19.485,46.587,36.235
C04233=1011.685,304.175,-163.974,-18.890,47.066,37.479
C04234=1011.577,304.411,-164.164,-18.265,47.545,38.750
C04235=1011.492,304.593,-164.314,-17.761,47.914,39.754
C04236=1011.408,304.775,-164.464,-17.237,48.283,40.777
C04237=1011.322,304.955,-164.615,-16.695,48.650,41.816
C04238=1011.237,305.135,-164.766,-16.132,49.015,42.875
C04239=1011.124,305.367,-164.964,-15.372,49.485,44.275
C04240=1011.011,305.599,-165.163,-14.578,49.950,45.708
C04241=1010.896,305.829,-165.363,-13.751,50.408,47.169
C04242=1010.781,306.057,-165.564,-12.888,50.859,48.662
C04243=1010.691,306.232,-165.720,-12.202,51.199,49.829
C04244=1010.601,306.406,-165.876,-11.496,51.534,51.012
C04245=1010.511,306.578,-166.033,-10.767,51.863,52.216
C04246=1010.419,306.751,-166.191,-10.018,52.186,53.439
C04247=1010.299,306.975,-166.399,-9.002,52.599,55.068
C04248=1010.178,307.197,-166.607,-7.948,53.000,56.733
C04249=1010.056,307.419,-166.818,-6.854,53.388,58.434
C04250=1009.933,307.639,-167.029,-5.724,53.761,60.165
C04251=1009.838,307.805,-167.191,-4.837,54.035,61.506
C04252=1009.743,307.970,-167.353,-3.930,54.299,62.863
C04253=1009.648,308.135,-167.516,-2.999,54.554,64.242
C04254=1009.552,308.299,-167.680,-2.047,54.798,65.640
C04255=1009.424,308.513,-167.897,-0.758,55.103,67.512
C04256=1009.295,308.727,-168.116,0.564,55.388,69.411
C04257=1009.166,308.939,-168.336,1.921,55.651,71.337
C04258=1009.034,309.149,-168.557,3.305,55.891,73.285
C04259=1008.940,309.300,-168.717,4.321,56.050,74.703
C04260=1008.844,309.450,-168.877,5.352,56.197,76.133
C04261=1008.743,309.598,-169.035,6.395,56.331,77.570
C04262=1008.635,309.745,-169.189,7.450,56.452,79.017
C04263=1008.522,309.890,-169.340,8.512,56.559,80.465
C04264=1008.403,310.034,-169.487,9.578,56.652,81.911
C04265=1008.279,310.175,-169.629,10.650,56.732,83.358
C04266=1008.149,310.314,-169.767,11.720,56.798,84.797
C04267=1008.449,310.434,-170.102,12.437,56.835,85.759
C04268=1008.596,310.280,-169.948,11.236,56.770,84.147
C04269=1008.738,310.122,-169.789,10.034,56.688,82.527
C04270=1008.873,309.962,-169.626,8.836,56.589,80.906
C04271=1009.001,309.800,-169.458,7.643,56.472,79.281
C04272=1009.114,309.646,-169.297,6.540,56.349,77.770
C04273=1009.221,309.491,-169.132,5.445,56.210,76.262
C04274=1009.321,309.335,-168.965,4.368,56.058,74.769
C04275=1009.421,309.177,-168.798,3.305,55.891,73.285
C04276=1009.551,308.967,-168.577,1.921,55.651,71.337
C04277=1009.681,308.754,-168.357,0.564,55.388,69.411
C04278=1009.810,308.541,-168.138,-0.758,55.103,67.512
C04279=1009.938,308.326,-167.921,-2.047,54.798,65.640
C04280=1010.034,308.162,-167.757,-2.999,54.554,64.242
C04281=1010.130,307.998,-167.594,-3.930,54.299,62.863
C04282=1010.225,307.833,-167.432,-4.837,54.035,61.506
C04283=1010.319,307.667,-167.270,-5.724,53.761,60.165
C04284=1010.442,307.446,-167.058,-6.854,53.388,58.434
C04285=1010.564,307.225,-166.848,-7.948,53.000,56.733
C04286=1010.686,307.002,-166.639,-9.002,52.599,55.068
C04287=1010.806,306.778,-166.432,-10.018,52.186,53.439
C04288=1010.897,306.606,-166.274,-10.767,51.863,52.216
C04289=1010.988,306.434,-166.117,-11.496,51.534,51.012
C04290=1011.077,306.260,-165.961,-12.202,51.199,49.829
C04291=1011.167,306.086,-165.805,-12.888,50.859,48.662
C04292=1011.283,305.857,-165.603,-13.751,50.408,47.169
C04293=1011.397,305.626,-165.404,-14.578,49.950,45.708
C04294=1011.510,305.396,-165.204,-15.372,49.485,44.275
C04295=1011.623,305.163,-165.007,-16.132,49.015,42.875
C04296=1011.709,304.983,-164.855,-16.695,48.650,41.816
C04297=1011.794,304.802,-164.704,-17.237,48.283,40.777
C04298=1011.879,304.621,-164.555,-17.761,47.914,39.754
C04299=1011.963,304.439,-164.406,-18.265,47.545,38.750
C04300=1012.071,304.203,-164.214,-18.890,47.066,37.479
C04301=1012.178,303.966,-164.025,-19.485,46.587,36.235
C04302=1012.284,303.727,-163.835,-20.052,46.107,35.019
C04303=1012.388,303.487,-163.649,-20.592,45.628,33.828
C04304=1012.469,303.299,-163.503,-20.996,45.254,32.916
C04305=1012.549,303.111,-163.359,-21.384,44.880,32.017
C04306=1012.629,302.922,-163.216,-21.757,44.508,31.133
C04307=1012.708,302.733,-163.073,-22.115,44.137,30.264
C04308=1012.809,302.490,-162.892,-22.552,43.665,29.173
C04309=1012.908,302.246,-162.712,-22.967,43.196,28.105
C04310=1013.005,302.001,-162.535,-23.359,42.732,27.060
C04311=1013.102,301.755,-162.357,-23.731,42.271,26.037
C04312=1013.178,301.560,-162.219,-24.010,41.911,25.245
C04313=1013.253,301.364,-162.081,-24.278,41.553,24.463
C04314=1013.327,301.169,-161.944,-24.533,41.199,23.695
C04315=1013.401,300.973,-161.808,-24.778,40.847,22.938
C04316=1013.494,300.724,-161.637,-25.071,40.409,21.999
C04317=1013.586,300.474,-161.468,-25.349,39.974,21.077
C04318=1013.676,300.223,-161.300,-25.611,39.544,20.170
///RCONF 0,0,0,0,1,0,0,0,0,0,0,0,0,0,0,0,0,0,0,0,0,0,0,0
C04319=1013.766,299.972,-161.133,-25.857,39.121,19.283
C04320=1013.836,299.771,-161.000,-26.044,38.788,18.586
C04321=1013.906,299.570,-160.870,-26.221,38.458,17.898
C04322=1013.976,299.368,-160.739,-26.391,38.132,17.220
C04323=1014.044,299.165,-160.610,-26.551,37.810,16.553
C04324=1014.129,298.911,-160.448,-26.741,37.414,15.733
C04325=1014.213,298.656,-160.289,-26.918,37.024,14.926
C04326=1014.297,298.400,-160.131,-27.085,36.640,14.133
C04327=1014.380,298.145,-159.974,-27.241,36.263,13.354
C04328=1014.445,297.938,-159.849,-27.359,35.964,12.737
C04329=1014.510,297.731,-159.724,-27.470,35.670,12.129
C04330=1014.575,297.523,-159.600,-27.576,35.380,11.529
C04331=1014.638,297.315,-159.477,-27.675,35.094,10.935
C04332=1014.717,297.057,-159.325,-27.790,34.746,10.213
C04333=1014.795,296.798,-159.175,-27.897,34.404,9.500
C04334=1014.871,296.538,-159.026,-27.996,34.068,8.799
C04335=1014.946,296.278,-158.879,-28.087,33.740,8.111
C04336=1015.007,296.066,-158.759,-28.156,33.478,7.560
C04337=1015.067,295.853,-158.641,-28.220,33.220,7.016
C04338=1015.127,295.641,-158.524,-28.280,32.966,6.479
C04339=1015.186,295.428,-158.407,-28.335,32.716,5.947
C04340=1015.258,295.166,-158.264,-28.398,32.417,5.306
C04341=1015.329,294.904,-158.123,-28.455,32.122,4.672
C04342=1015.399,294.640,-157.983,-28.506,31.835,4.050
C04343=1015.469,294.377,-157.844,-28.552,31.552,3.436
C04344=1015.524,294.160,-157.730,-28.586,31.327,2.940
C04345=1015.580,293.944,-157.618,-28.617,31.104,2.450
C04346=1015.636,293.726,-157.507,-28.645,30.886,1.967
C04347=1015.690,293.509,-157.396,-28.669,30.673,1.490
C04348=1015.755,293.243,-157.263,-28.695,30.417,0.916
C04349=1015.820,292.978,-157.130,-28.717,30.168,0.353
C04350=1015.884,292.711,-156.998,-28.736,29.926,-0.203
C04351=1015.948,292.445,-156.867,-28.751,29.688,-0.751
C04352=1015.999,292.224,-156.761,-28.761,29.494,-1.200
C04353=1016.051,292.004,-156.654,-28.768,29.306,-1.642
C04354=1016.101,291.783,-156.549,-28.773,29.120,-2.080
C04355=1016.152,291.561,-156.443,-28.777,28.937,-2.514
C04356=1016.211,291.293,-156.318,-28.778,28.722,-3.030
C04357=1016.271,291.025,-156.193,-28.777,28.512,-3.541
C04358=1016.329,290.756,-156.069,-28.773,28.305,-4.046
C04359=1016.387,290.487,-155.946,-28.767,28.103,-4.544
C04360=1016.434,290.263,-155.844,-28.760,27.939,-4.952
C04361=1016.482,290.039,-155.745,-28.752,27.779,-5.357
C04362=1016.528,289.815,-155.644,-28.742,27.622,-5.757
C04363=1016.574,289.589,-155.545,-28.730,27.467,-6.153
C04364=1016.628,289.319,-155.426,-28.715,27.285,-6.624
C04365=1016.682,289.049,-155.310,-28.698,27.109,-7.088
C04366=1016.735,288.778,-155.193,-28.679,26.937,-7.545
C04367=1016.787,288.507,-155.077,-28.659,26.767,-7.999
C04368=1016.832,288.280,-154.982,-28.641,26.630,-8.372
C04369=1016.875,288.052,-154.887,-28.622,26.495,-8.743
C04370=1016.917,287.824,-154.792,-28.602,26.363,-9.109
C04371=1016.959,287.596,-154.698,-28.581,26.233,-9.471
C04372=1017.008,287.325,-154.587,-28.555,26.082,-9.899
C04373=1017.057,287.052,-154.476,-28.527,25.936,-10.320
C04374=1017.105,286.780,-154.368,-28.499,25.792,-10.737
C04375=1017.153,286.507,-154.259,-28.470,25.652,-11.148
C04376=1017.192,286.277,-154.168,-28.444,25.537,-11.492
C04377=1017.231,286.047,-154.078,-28.418,25.425,-11.832
C04378=1017.270,285.816,-153.988,-28.391,25.314,-12.171
C04379=1017.309,285.586,-153.900,-28.364,25.204,-12.507
C04380=1017.353,285.313,-153.795,-28.330,25.079,-12.901
C04381=1017.397,285.039,-153.692,-28.296,24.956,-13.292
C04382=1017.440,284.766,-153.589,-28.261,24.835,-13.680
C04383=1017.484,284.491,-153.488,-28.226,24.716,-14.065
C04384=1017.520,284.259,-153.402,-28.195,24.619,-14.388
C04385=1017.555,284.026,-153.317,-28.164,24.524,-14.708
C04386=1017.590,283.793,-153.232,-28.132,24.429,-15.026
C04387=1017.624,283.560,-153.148,-28.100,24.338,-15.343
C04388=1017.664,283.286,-153.050,-28.062,24.232,-15.713
C04389=1017.704,283.012,-152.953,-28.023,24.128,-16.079
C04390=1017.743,282.736,-152.857,-27.984,24.027,-16.441
C04391=1017.781,282.461,-152.761,-27.945,23.929,-16.801
C04392=1017.814,282.226,-152.681,-27.911,23.848,-17.104
C04393=1017.845,281.991,-152.601,-27.877,23.768,-17.406
C04394=1017.876,281.756,-152.521,-27.842,23.690,-17.706
C04395=1017.908,281.521,-152.442,-27.807,23.613,-18.004
C04396=1017.943,281.245,-152.351,-27.766,23.526,-18.349
C04397=1017.979,280.970,-152.259,-27.725,23.440,-18.691
C04398=1018.013,280.693,-152.169,-27.684,23.357,-19.031
C04399=1018.047,280.418,-152.079,-27.642,23.276,-19.367
C04400=1018.076,280.181,-152.003,-27.606,23.208,-19.653
C04401=1018.104,279.944,-151.929,-27.570,23.142,-19.936
C04402=1018.132,279.707,-151.854,-27.534,23.078,-20.218
C04403=1018.160,279.470,-151.779,-27.498,23.014,-20.499
C04404=1018.192,279.194,-151.693,-27.456,22.942,-20.824
C04405=1018.223,278.917,-151.607,-27.413,22.873,-21.147
C04406=1018.254,278.641,-151.523,-27.370,22.804,-21.469
C04407=1018.283,278.364,-151.440,-27.327,22.737,-21.789
C04408=1018.308,278.125,-151.369,-27.290,22.681,-22.062
C04409=1018.334,277.887,-151.298,-27.252,22.626,-22.334
C04410=1018.359,277.648,-151.228,-27.215,22.573,-22.606
C04411=1018.383,277.409,-151.158,-27.177,22.521,-22.877
C04412=1018.410,277.132,-151.078,-27.134,22.462,-23.186
C04413=1018.437,276.855,-150.998,-27.090,22.404,-23.496
C04414=1018.464,276.578,-150.919,-27.046,22.349,-23.804
C04415=1018.490,276.300,-150.842,-27.003,22.295,-24.109
C04416=1018.512,276.061,-150.775,-26.965,22.250,-24.373
C04417=1018.533,275.820,-150.709,-26.927,22.204,-24.635
C04418=1018.555,275.579,-150.643,-26.889,22.162,-24.896
C04419=1018.576,275.340,-150.578,-26.851,22.119,-25.156
C04420=1018.600,275.062,-150.503,-26.807,22.073,-25.453
C04421=1018.623,274.784,-150.430,-26.763,22.027,-25.750
C04422=1018.645,274.506,-150.357,-26.720,21.983,-26.043
C04423=1018.668,274.228,-150.283,-26.676,21.940,-26.336
C04424=1018.687,273.987,-150.222,-26.638,21.904,-26.589
C04425=1018.705,273.745,-150.159,-26.600,21.869,-26.841
C04426=1018.723,273.503,-150.098,-26.562,21.835,-27.092
C04427=1018.742,273.262,-150.037,-26.525,21.803,-27.342
C04428=1018.760,272.984,-149.968,-26.481,21.766,-27.626
C04429=1018.780,272.705,-149.900,-26.438,21.731,-27.910
C04430=1018.799,272.428,-149.832,-26.395,21.697,-28.194
C04431=1018.817,272.149,-149.766,-26.351,21.664,-28.476
C04432=1018.833,271.907,-149.707,-26.314,21.637,-28.720
C04433=1018.849,271.664,-149.650,-26.276,21.610,-28.964
C04434=1018.864,271.421,-149.593,-26.238,21.585,-29.208
C04435=1018.878,271.178,-149.537,-26.201,21.560,-29.450
C04436=1018.895,270.899,-149.473,-26.158,21.533,-29.728
C04437=1018.910,270.621,-149.409,-26.115,21.507,-30.003
C04438=1018.925,270.343,-149.347,-26.072,21.483,-30.277
C04439=1018.941,270.064,-149.286,-26.030,21.459,-30.551
C04440=1018.953,269.821,-149.232,-25.992,21.439,-30.791
C04441=1018.965,269.577,-149.179,-25.955,21.420,-31.029
C04442=1018.976,269.333,-149.126,-25.918,21.402,-31.266
C04443=1018.988,269.088,-149.074,-25.881,21.386,-31.502
C04444=1019.000,268.809,-149.016,-25.839,21.367,-31.772
C04445=1019.012,268.531,-148.958,-25.797,21.350,-32.039
C04446=1019.024,268.252,-148.900,-25.755,21.333,-32.307
C04447=1019.036,267.974,-148.844,-25.714,21.319,-32.571
C04448=1019.044,267.728,-148.795,-25.677,21.306,-32.805
C04449=1019.053,267.484,-148.746,-25.641,21.295,-33.037
C04450=1019.063,267.238,-148.698,-25.604,21.284,-33.269
C04451=1019.071,266.993,-148.650,-25.568,21.275,-33.499
C04452=1019.079,266.714,-148.597,-25.527,21.264,-33.760
C04453=1019.088,266.435,-148.544,-25.487,21.254,-34.021
C04454=1019.096,266.157,-148.492,-25.446,21.246,-34.279
C04455=1019.104,265.878,-148.441,-25.406,21.239,-34.538
C04456=1019.110,265.632,-148.396,-25.370,21.233,-34.766
C04457=1019.116,265.386,-148.351,-25.335,21.229,-34.991
C04458=1019.122,265.139,-148.307,-25.300,21.225,-35.219
C04459=1019.127,264.893,-148.264,-25.265,21.221,-35.444
C04460=1019.132,264.614,-148.216,-25.226,21.219,-35.699
C04461=1019.137,264.335,-148.168,-25.186,21.216,-35.954
C04462=1019.142,264.056,-148.121,-25.147,21.215,-36.207
C04463=1019.146,263.776,-148.074,-25.108,21.216,-36.459
C04464=1019.149,263.530,-148.034,-25.074,21.217,-36.681
C04465=1019.152,263.283,-147.994,-25.040,21.218,-36.903
C04466=1019.155,263.036,-147.955,-25.006,21.220,-37.124
C04467=1019.157,262.790,-147.915,-24.973,21.223,-37.345
C04468=1019.158,262.510,-147.872,-24.935,21.227,-37.593
C04469=1019.160,262.231,-147.829,-24.897,21.233,-37.842
C04470=1019.161,261.951,-147.787,-24.860,21.238,-38.090
C04471=1019.163,261.672,-147.746,-24.823,21.245,-38.337
C04472=1019.162,261.424,-147.710,-24.790,21.251,-38.554
C04473=1019.163,261.177,-147.674,-24.758,21.259,-38.770
C04474=1019.162,260.930,-147.639,-24.725,21.267,-38.988
C04475=1019.161,260.682,-147.604,-24.693,21.275,-39.204
C04476=1019.160,260.402,-147.565,-24.658,21.287,-39.446
C04477=1019.158,260.122,-147.528,-24.622,21.298,-39.688
C04478=1019.156,259.843,-147.491,-24.587,21.310,-39.930
C04479=1019.153,259.563,-147.454,-24.551,21.322,-40.171
C04480=1019.136,258.328,-147.300,-24.430,21.375,-41.012
C04481=1019.131,258.084,-147.271,-24.430,21.375,-41.014
C04482=1019.128,257.840,-147.242,-24.429,21.375,-41.018
C04483=1019.125,257.596,-147.212,-24.429,21.376,-41.019
C04484=1019.122,257.353,-147.183,-24.429,21.376,-41.021
C04485=1019.118,257.110,-147.155,-24.428,21.375,-41.025
C04486=1019.115,256.866,-147.125,-24.428,21.376,-41.027
C04487=1019.111,256.623,-147.095,-24.428,21.377,-41.029
C04488=1019.108,256.375,-147.067,-24.427,21.376,-41.032
C04489=1019.105,256.127,-147.036,-24.427,21.376,-41.034
C04490=1019.101,255.878,-147.007,-24.426,21.376,-41.037
C04491=1019.098,255.630,-146.977,-24.426,21.377,-41.040
C04492=1019.094,255.382,-146.948,-24.426,21.377,-41.042
C04493=1019.090,255.134,-146.918,-24.425,21.377,-41.045
C04494=1019.087,254.885,-146.889,-24.425,21.377,-41.047
C04495=1019.084,254.638,-146.859,-24.425,21.377,-41.049
C04496=1019.081,254.389,-146.829,-24.424,21.378,-41.052
C04497=1019.077,254.141,-146.801,-24.424,21.378,-41.054
C04498=1019.074,253.893,-146.770,-24.424,21.378,-41.058
C04499=1019.071,253.645,-146.741,-24.423,21.378,-41.060
C04500=1019.067,253.396,-146.711,-24.423,21.378,-41.061
C04501=1019.063,253.148,-146.682,-24.423,21.378,-41.065
C04502=1019.061,252.899,-146.652,-24.422,21.379,-41.067
C04503=1019.057,252.651,-146.622,-24.422,21.379,-41.069
C04504=1019.053,252.403,-146.594,-24.421,21.378,-41.072
C04505=1019.050,252.154,-146.564,-24.421,21.379,-41.074
C04506=1019.047,251.907,-146.534,-24.421,21.380,-41.076
C04507=1019.044,251.659,-146.505,-24.421,21.380,-41.078
C04508=1019.040,251.415,-146.476,-24.420,21.380,-41.082
C04509=1019.037,251.172,-146.447,-24.420,21.380,-41.084
C04510=1019.035,250.929,-146.418,-24.420,21.380,-41.085
C04511=1019.031,250.685,-146.390,-24.419,21.380,-41.089
C04512=1019.028,250.441,-146.361,-24.419,21.380,-41.091
C04513=1019.024,250.198,-146.333,-24.419,21.381,-41.093
C04514=1019.022,249.955,-146.304,-24.418,21.381,-41.095
C04515=1019.018,249.711,-146.274,-24.418,21.381,-41.098
C04516=1019.015,249.463,-146.246,-24.418,21.381,-41.100
C04517=1019.011,249.215,-146.216,-24.417,21.381,-41.102
C04518=1019.009,248.966,-146.187,-24.417,21.381,-41.104
C04519=1019.005,248.719,-146.158,-24.417,21.381,-41.107
C04520=1019.002,248.470,-146.128,-24.416,21.381,-41.109
C04521=1018.999,248.222,-146.099,-24.416,21.382,-41.111
C04522=1018.996,247.974,-146.070,-24.416,21.382,-41.113
C04523=1018.992,247.725,-146.041,-24.415,21.382,-41.117
C04524=1018.989,247.477,-146.012,-24.415,21.382,-41.118
C04525=1018.987,247.229,-145.982,-24.415,21.382,-41.120
C04526=1018.983,246.980,-145.953,-24.414,21.383,-41.122
C04527=1018.980,246.732,-145.924,-24.414,21.382,-41.126
C04528=1018.977,246.484,-145.895,-24.414,21.382,-41.127
C04529=1018.974,246.236,-145.866,-24.413,21.383,-41.129
C04530=1018.971,245.987,-145.837,-24.413,21.384,-41.132
C04531=1018.967,245.739,-145.808,-24.413,21.384,-41.134
C04532=1018.965,245.491,-145.778,-24.412,21.384,-41.137
C04533=1018.962,245.243,-145.750,-24.412,21.384,-41.139
C04534=1018.958,244.994,-145.720,-24.412,21.384,-41.141
C04535=1018.955,244.746,-145.691,-24.412,21.384,-41.143
C04536=1018.952,244.503,-145.663,-24.411,21.384,-41.144
C04537=1018.949,244.260,-145.634,-24.411,21.384,-41.148
C04538=1018.946,244.016,-145.606,-24.411,21.384,-41.150
C04539=1018.943,243.773,-145.577,-24.410,21.384,-41.151
C04540=1018.939,243.530,-145.549,-24.410,21.385,-41.153
C04541=1018.937,243.287,-145.520,-24.410,21.385,-41.155
C04542=1018.934,243.044,-145.492,-24.410,21.385,-41.157
C04543=1018.931,242.800,-145.464,-24.409,21.385,-41.159
C04544=1018.928,242.552,-145.435,-24.409,21.385,-41.162
C04545=1018.925,242.303,-145.405,-24.408,21.385,-41.164
C04546=1018.922,242.056,-145.377,-24.408,21.385,-41.166
C04547=1018.919,241.808,-145.348,-24.408,21.386,-41.168
C04548=1018.916,241.559,-145.319,-24.408,21.386,-41.170
C04549=1018.913,241.311,-145.290,-24.407,21.386,-41.172
C04550=1018.910,241.062,-145.261,-24.407,21.386,-41.174
C04551=1018.907,240.814,-145.232,-24.407,21.386,-41.177
C04552=1018.904,240.566,-145.203,-24.406,21.386,-41.179
C04553=1018.901,240.317,-145.174,-24.406,21.386,-41.181
C04554=1018.898,240.069,-145.146,-24.406,21.386,-41.183
C04555=1018.896,239.821,-145.116,-24.406,21.387,-41.184
C04556=1018.892,239.573,-145.088,-24.405,21.387,-41.186
C04557=1018.889,239.324,-145.059,-24.405,21.387,-41.188
C04558=1018.887,239.076,-145.030,-24.405,21.387,-41.190
C04559=1018.884,238.828,-145.001,-24.405,21.388,-41.192
C04560=1018.881,238.579,-144.973,-24.404,21.387,-41.195
C04561=1018.878,238.331,-144.944,-24.404,21.387,-41.197
C04562=1018.875,238.083,-144.915,-24.403,21.388,-41.199
C04563=1018.873,237.834,-144.886,-24.403,21.388,-41.201
C04564=1018.869,237.591,-144.858,-24.403,21.388,-41.203
C04565=1018.866,237.348,-144.831,-24.403,21.388,-41.205
C04566=1018.864,237.105,-144.802,-24.402,21.388,-41.207
C04567=1018.860,236.861,-144.774,-24.402,21.389,-41.209
C04568=1018.858,236.618,-144.746,-24.402,21.389,-41.210
C04569=1018.855,236.375,-144.717,-24.402,21.389,-41.212
C04570=1018.853,236.132,-144.690,-24.401,21.389,-41.214
C04571=1018.850,235.889,-144.662,-24.401,21.390,-41.216
C04572=1018.847,235.641,-144.633,-24.401,21.389,-41.218
C04573=1018.844,235.393,-144.604,-24.401,21.389,-41.219
C04574=1018.841,235.144,-144.576,-24.400,21.389,-41.221
C04575=1018.838,234.896,-144.547,-24.400,21.390,-41.223
C04576=1018.836,234.647,-144.518,-24.400,21.390,-41.225
C04577=1018.833,234.399,-144.490,-24.400,21.390,-41.227
C04578=1018.830,234.151,-144.462,-24.399,21.390,-41.229
C04579=1018.827,233.903,-144.432,-24.399,21.390,-41.231
C04580=1018.824,233.654,-144.404,-24.399,21.391,-41.233
C04581=1018.822,233.405,-144.375,-24.399,21.391,-41.234
C04582=1018.819,233.158,-144.347,-24.398,21.391,-41.236
C04583=1018.816,232.909,-144.319,-24.398,21.390,-41.238
C04584=1018.814,232.661,-144.290,-24.398,21.391,-41.240
C04585=1018.811,232.412,-144.262,-24.397,21.391,-41.242
C04586=1018.808,232.164,-144.233,-24.397,21.391,-41.243
C04587=1018.805,231.915,-144.204,-24.397,21.391,-41.245
C04588=1018.803,231.667,-144.176,-24.397,21.392,-41.247
C04589=1018.801,231.419,-144.147,-24.396,21.392,-41.249
C04590=1018.798,231.171,-144.119,-24.396,21.392,-41.251
C04591=1018.795,230.922,-144.091,-24.396,21.391,-41.252
C04592=1018.792,230.679,-144.063,-24.396,21.392,-41.254
C04593=1018.790,230.437,-144.035,-24.395,21.392,-41.256
C04594=1018.787,230.193,-144.007,-24.395,21.392,-41.258
C04595=1018.785,229.950,-143.979,-24.395,21.392,-41.260
C04596=1018.782,229.707,-143.952,-24.395,21.392,-41.262
C04597=1018.779,229.464,-143.924,-24.394,21.392,-41.263
C04598=1018.777,229.221,-143.895,-24.394,21.392,-41.265
C04599=1018.774,228.978,-143.868,-24.394,21.393,-41.266
C04600=1018.771,228.730,-143.840,-24.394,21.393,-41.267
C04601=1018.769,228.481,-143.812,-24.394,21.393,-41.269
C04602=1018.766,228.233,-143.784,-24.393,21.394,-41.271
C04603=1018.764,227.985,-143.754,-24.393,21.393,-41.273
C04604=1018.761,227.736,-143.726,-24.393,21.393,-41.275
C04605=1018.758,227.488,-143.698,-24.393,21.393,-41.276
C04606=1018.756,227.239,-143.670,-24.392,21.394,-41.278
C04607=1018.754,226.991,-143.642,-24.392,21.394,-41.280
C04608=1018.751,226.742,-143.614,-24.392,21.393,-41.282
C04609=1018.748,226.494,-143.585,-24.391,21.393,-41.284
C04610=1018.746,226.246,-143.557,-24.391,21.394,-41.285
C04611=1018.743,225.998,-143.529,-24.391,21.395,-41.286
C04612=1018.741,225.749,-143.500,-24.391,21.395,-41.288
C04613=1018.738,225.501,-143.472,-24.391,21.394,-41.289
C04614=1018.735,225.252,-143.444,-24.390,21.394,-41.291
C04615=1018.734,225.004,-143.416,-24.390,21.395,-41.293
C04616=1018.731,224.756,-143.388,-24.390,21.395,-41.295
C04617=1018.729,224.507,-143.359,-24.390,21.395,-41.297
C04618=1018.726,224.259,-143.332,-24.389,21.394,-41.298
C04619=1018.723,224.010,-143.304,-24.389,21.395,-41.300
C04620=1018.721,223.768,-143.275,-24.389,21.395,-41.300
C04621=1018.718,223.525,-143.248,-24.389,21.396,-41.302
C04622=1018.716,223.282,-143.220,-24.389,21.396,-41.304
C04623=1018.713,223.039,-143.193,-24.388,21.395,-41.306
C04624=1018.712,222.795,-143.166,-24.388,21.395,-41.308
C04625=1018.709,222.553,-143.139,-24.388,21.396,-41.309
C04626=1018.707,222.310,-143.111,-24.388,21.397,-41.310
C04627=1018.705,222.067,-143.083,-24.388,21.396,-41.311
C04628=1018.702,221.818,-143.055,-24.387,21.396,-41.313
C04629=1018.700,221.570,-143.027,-24.387,21.396,-41.315
C04630=1018.697,221.322,-142.999,-24.387,21.397,-41.317
C04631=1018.695,221.074,-142.971,-24.386,21.396,-41.318
C04632=1018.692,220.825,-142.943,-24.386,21.396,-41.320
C04633=1018.690,220.577,-142.915,-24.386,21.397,-41.321
C04634=1018.687,220.328,-142.887,-24.386,21.397,-41.323
C04635=1018.685,220.080,-142.859,-24.386,21.397,-41.324
C04636=1018.683,219.831,-142.830,-24.385,21.397,-41.326
C04637=1018.681,219.584,-142.803,-24.385,21.397,-41.328
C04638=1018.678,219.334,-142.775,-24.385,21.397,-41.330
C04639=1018.676,219.086,-142.747,-24.385,21.397,-41.330
C04640=1018.673,218.838,-142.719,-24.385,21.397,-41.332
C04641=1018.671,218.590,-142.691,-24.384,21.398,-41.333
C04642=1018.669,218.341,-142.663,-24.384,21.398,-41.335
C04643=1018.666,218.093,-142.635,-24.384,21.397,-41.337
C04644=1018.665,217.844,-142.607,-24.384,21.397,-41.339
C04645=1018.662,217.595,-142.579,-24.384,21.398,-41.339
C04646=1018.660,217.348,-142.551,-24.383,21.399,-41.341
C04647=1018.658,217.099,-142.523,-24.383,21.398,-41.342
C04648=1018.654,216.789,-142.489,-24.383,21.398,-41.344
C04649=1018.652,216.479,-142.454,-24.383,21.398,-41.346
C04650=1018.648,216.168,-142.419,-24.382,21.399,-41.348
C04651=1018.646,215.858,-142.384,-24.382,21.399,-41.350
C04652=1018.644,215.610,-142.356,-24.382,21.399,-41.352
C04653=1018.643,215.361,-142.329,-24.382,21.398,-41.353
C04654=1018.640,215.112,-142.301,-24.382,21.399,-41.354
C04655=1018.637,214.864,-142.273,-24.381,21.400,-41.356
C04656=1018.635,214.615,-142.245,-24.381,21.400,-41.358
C04657=1018.633,214.367,-142.217,-24.381,21.399,-41.359
C04658=1018.631,214.119,-142.190,-24.381,21.399,-41.361
C04659=1018.629,213.870,-142.162,-24.381,21.400,-41.361
C04660=1018.626,213.622,-142.134,-24.380,21.400,-41.363
C04661=1018.625,213.374,-142.106,-24.380,21.400,-41.365
C04662=1018.623,213.125,-142.079,-24.380,21.400,-41.366
C04663=1018.620,212.876,-142.051,-24.379,21.399,-41.368
C04664=1018.618,212.628,-142.023,-24.380,21.400,-41.368
C04665=1018.616,212.380,-141.995,-24.379,21.400,-41.370
C04666=1018.613,212.131,-141.967,-24.379,21.400,-41.372
C04667=1018.612,211.882,-141.940,-24.379,21.400,-41.374
C04668=1018.609,211.634,-141.912,-24.379,21.401,-41.374
C04669=1018.607,211.386,-141.885,-24.379,21.401,-41.376
C04670=1018.605,211.137,-141.856,-24.378,21.400,-41.377
C04671=1018.603,210.888,-141.829,-24.378,21.401,-41.379
C04672=1018.601,210.538,-141.790,-24.378,21.401,-41.381
C04673=1018.598,210.188,-141.751,-24.377,21.401,-41.383
C04674=1018.595,209.945,-141.724,-24.377,21.401,-41.383
C04675=1018.593,209.702,-141.697,-24.377,21.401,-41.385
C04676=1018.591,209.459,-141.670,-24.377,21.402,-41.387
C04677=1018.589,209.218,-141.643,-24.377,21.401,-41.388
C04678=1018.587,208.974,-141.617,-24.377,21.402,-41.389
C04679=1018.585,208.732,-141.589,-24.376,21.402,-41.391
C04680=1018.583,208.488,-141.562,-24.376,21.401,-41.392
C04681=1018.581,208.246,-141.535,-24.376,21.402,-41.392
C04682=1018.579,207.997,-141.508,-24.376,21.402,-41.394
C04683=1018.577,207.749,-141.480,-24.376,21.402,-41.396
C04684=1018.575,207.501,-141.453,-24.375,21.402,-41.398
C04685=1018.573,207.253,-141.425,-24.375,21.402,-41.398
C04686=1018.572,207.004,-141.398,-24.375,21.402,-41.399
C04687=1018.569,206.755,-141.370,-24.375,21.402,-41.401
C04688=1018.567,206.507,-141.342,-24.375,21.402,-41.401
C04689=1018.565,206.258,-141.315,-24.375,21.403,-41.403
C04690=1018.563,206.010,-141.287,-24.374,21.403,-41.405
C04691=1018.562,205.761,-141.260,-24.374,21.402,-41.407
C04692=1018.559,205.513,-141.233,-24.374,21.403,-41.407
C04693=1018.557,205.265,-141.205,-24.374,21.403,-41.409
C04694=1018.556,205.016,-141.178,-24.373,21.403,-41.410
C04695=1018.554,204.768,-141.151,-24.374,21.404,-41.411
C04696=1018.552,204.519,-141.124,-24.373,21.403,-41.412
C04697=1018.550,204.271,-141.095,-24.373,21.403,-41.414
C04698=1018.547,204.022,-141.068,-24.373,21.404,-41.415
C04699=1018.546,203.773,-141.040,-24.373,21.403,-41.416
C04700=1018.540,202.557,-140.904,-24.425,21.378,-41.051
C04701=1018.538,202.170,-140.861,-24.424,21.378,-41.052
C04702=1018.537,201.820,-140.822,-24.424,21.378,-41.054
C04703=1018.538,201.469,-140.783,-24.424,21.378,-41.058
C04704=1018.538,201.062,-140.738,-24.423,21.379,-41.060
C04705=1018.538,200.836,-140.714,-24.423,21.378,-41.061
C04706=1018.539,200.606,-140.688,-24.423,21.378,-41.063
C04707=1018.539,200.383,-140.664,-24.423,21.378,-41.065
C04708=1018.539,200.170,-140.640,-24.423,21.378,-41.065
C04709=1018.539,199.770,-140.596,-24.422,21.379,-41.069
C04710=1018.540,199.381,-140.554,-24.422,21.379,-41.071
C04711=1018.541,198.983,-140.510,-24.421,21.379,-41.074
C04712=1018.542,198.581,-140.467,-24.421,21.379,-41.076
C04713=1018.542,198.180,-140.422,-24.421,21.380,-41.078
C04714=1018.543,197.778,-140.379,-24.420,21.380,-41.082
C04715=1018.543,197.378,-140.335,-24.420,21.380,-41.084
C04716=1018.544,196.977,-140.291,-24.419,21.380,-41.087
C04717=1018.545,196.576,-140.247,-24.419,21.380,-41.089
C04718=1018.546,196.174,-140.203,-24.419,21.381,-41.091
C04719=1018.546,195.773,-140.160,-24.418,21.380,-41.094
C04720=1018.547,195.372,-140.116,-24.418,21.381,-41.097
C04721=1018.547,194.971,-140.072,-24.418,21.381,-41.100
C04722=1018.548,194.570,-140.029,-24.417,21.381,-41.102
C04723=1018.549,194.169,-139.984,-24.417,21.381,-41.105
C04724=1018.550,193.767,-139.941,-24.417,21.382,-41.108
C04725=1018.551,193.366,-139.898,-24.416,21.382,-41.109
C04726=1018.551,192.966,-139.854,-24.416,21.382,-41.113
C04727=1018.552,192.564,-139.810,-24.415,21.382,-41.115
C04728=1018.553,192.163,-139.767,-24.415,21.382,-41.118
C04729=1018.554,191.762,-139.724,-24.415,21.382,-41.120
C04730=1018.555,191.360,-139.680,-24.414,21.382,-41.124
C04731=1018.556,190.960,-139.636,-24.414,21.383,-41.126
C04732=1018.556,190.559,-139.593,-24.414,21.383,-41.128
C04733=1018.557,190.157,-139.549,-24.413,21.383,-41.131
C04734=1018.558,189.756,-139.506,-24.413,21.383,-41.133
C04735=1018.559,189.355,-139.463,-24.412,21.384,-41.137
C04736=1018.560,188.955,-139.420,-24.412,21.384,-41.139
C04737=1018.561,188.553,-139.376,-24.412,21.384,-41.141
C04738=1018.561,188.153,-139.332,-24.411,21.384,-41.144
C04739=1018.562,187.752,-139.289,-24.411,21.385,-41.146
C04740=1018.563,187.350,-139.246,-24.411,21.384,-41.150
C04741=1018.564,186.950,-139.203,-24.410,21.384,-41.151
C04742=1018.565,186.549,-139.159,-24.410,21.384,-41.155
C04743=1018.565,186.147,-139.116,-24.410,21.385,-41.157
C04744=1018.567,185.746,-139.072,-24.409,21.385,-41.159
C04745=1018.568,185.345,-139.029,-24.409,21.385,-41.162
C04746=1018.569,184.944,-138.986,-24.409,21.386,-41.165
C04747=1018.570,184.543,-138.943,-24.408,21.386,-41.168
C04748=1018.570,184.143,-138.900,-24.408,21.386,-41.170
C04749=1018.571,183.741,-138.857,-24.407,21.386,-41.172
C04750=1018.572,183.341,-138.814,-24.407,21.386,-41.176
C04751=1018.574,182.939,-138.771,-24.407,21.387,-41.177
C04752=1018.575,182.539,-138.728,-24.406,21.386,-41.181
C04753=1018.576,182.137,-138.685,-24.406,21.387,-41.183
C04754=1018.577,181.737,-138.642,-24.405,21.387,-41.186
C04755=1018.578,181.336,-138.599,-24.405,21.387,-41.188
C04756=1018.579,180.935,-138.556,-24.405,21.387,-41.190
C04757=1018.580,180.534,-138.513,-24.404,21.388,-41.194
C04758=1018.581,180.133,-138.470,-24.404,21.388,-41.196
C04759=1018.582,179.732,-138.427,-24.403,21.388,-41.199
C04760=1018.584,179.331,-138.384,-24.403,21.388,-41.201
C04761=1018.584,178.931,-138.342,-24.403,21.388,-41.205
C04762=1018.585,178.530,-138.298,-24.402,21.388,-41.207
C04763=1018.586,178.129,-138.256,-24.402,21.389,-41.209
C04764=1018.588,177.728,-138.213,-24.402,21.389,-41.212
C04765=1018.589,177.327,-138.170,-24.401,21.389,-41.214
C04766=1018.589,176.927,-138.128,-24.401,21.389,-41.218
C04767=1018.591,176.526,-138.085,-24.401,21.389,-41.219
C04768=1018.592,176.125,-138.042,-24.400,21.390,-41.223
C04769=1018.594,175.725,-137.999,-24.400,21.390,-41.225
C04770=1018.594,175.323,-137.956,-24.400,21.390,-41.227
C04771=1018.595,174.923,-137.914,-24.399,21.390,-41.231
C04772=1018.597,174.522,-137.872,-24.399,21.391,-41.233
C04773=1018.598,174.122,-137.829,-24.398,21.390,-41.236
C04774=1018.599,173.721,-137.786,-24.398,21.390,-41.238
C04775=1018.600,173.320,-137.744,-24.397,21.391,-41.242
C04776=1018.602,172.920,-137.701,-24.397,21.391,-41.243
C04777=1018.603,172.519,-137.658,-24.397,21.391,-41.247
C04778=1018.604,172.119,-137.616,-24.396,21.392,-41.249
C04779=1018.605,171.718,-137.574,-24.396,21.392,-41.251
C04780=1018.607,171.317,-137.531,-24.396,21.392,-41.254
C04781=1018.608,170.917,-137.489,-24.395,21.392,-41.256
C04782=1018.609,170.516,-137.446,-24.395,21.392,-41.260
C04783=1018.609,170.116,-137.404,-24.395,21.392,-41.262
C04784=1018.611,169.715,-137.361,-24.394,21.392,-41.265
C04785=1018.612,169.314,-137.319,-24.394,21.393,-41.267
C04786=1018.614,168.915,-137.277,-24.393,21.393,-41.271
C04787=1018.615,168.514,-137.234,-24.393,21.393,-41.273
C04788=1018.616,168.113,-137.192,-24.393,21.394,-41.275
C04789=1018.618,167.712,-137.150,-24.392,21.394,-41.278
C04790=1018.618,167.312,-137.107,-24.392,21.394,-41.280
C04791=1018.620,166.912,-137.065,-24.391,21.393,-41.284
C04792=1018.621,166.511,-137.023,-24.391,21.395,-41.286
C04793=1018.622,166.111,-136.980,-24.391,21.394,-41.289
C04794=1018.624,165.711,-136.939,-24.390,21.394,-41.291
C04795=1018.625,165.310,-136.896,-24.390,21.395,-41.295
C04796=1018.626,164.910,-136.854,-24.390,21.395,-41.297
C04797=1018.628,164.510,-136.812,-24.389,21.395,-41.300
C04798=1018.629,164.123,-136.771,-24.389,21.395,-41.302
C04799=1018.630,163.934,-136.752,-24.389,21.395,-41.304
C04800=1018.632,163.522,-136.708,-24.388,21.396,-41.306
C04801=1018.632,163.287,-136.684,-24.388,21.395,-41.308
C04802=1018.633,163.033,-136.657,-24.388,21.396,-41.309
C04803=1018.634,162.770,-136.629,-24.388,21.396,-41.311
C04804=1018.635,162.501,-136.602,-24.387,21.396,-41.313
C04805=1018.636,162.230,-136.572,-24.387,21.396,-41.315
C04806=1018.636,161.960,-136.544,-24.387,21.397,-41.317
C04807=1018.637,161.698,-136.517,-24.387,21.397,-41.319
C04808=1018.638,161.447,-136.490,-24.386,21.396,-41.320
C04809=1018.638,161.209,-136.465,-24.386,21.396,-41.322
C04810=1018.639,160.985,-136.442,-24.386,21.397,-41.324
C04811=1018.641,160.771,-136.420,-24.386,21.397,-41.325
C04812=1018.642,160.367,-136.377,-24.385,21.397,-41.328
C04813=1018.643,159.970,-136.336,-24.385,21.397,-41.330
C04814=1018.644,159.569,-136.293,-24.384,21.398,-41.333
C04815=1018.650,159.168,-136.255,-24.384,21.398,-41.335
C04816=1018.656,158.767,-136.215,-24.384,21.397,-41.339
C04817=1018.662,158.366,-136.176,-24.383,21.399,-41.341
C04818=1018.668,157.963,-136.137,-24.383,21.398,-41.344
C04819=1018.675,157.559,-136.098,-24.383,21.398,-41.346
C04820=1018.680,157.155,-136.058,-24.382,21.399,-41.350
C04821=1018.687,156.750,-136.019,-24.382,21.399,-41.352
C04822=1018.693,156.345,-135.979,-24.381,21.399,-41.355
C04823=1018.699,155.937,-135.939,-24.381,21.400,-41.358
C04824=1018.705,155.529,-135.901,-24.381,21.399,-41.361
C04825=1018.711,155.121,-135.860,-24.380,21.400,-41.363
C04826=1018.717,154.711,-135.821,-24.380,21.400,-41.366
C04827=1018.723,154.301,-135.780,-24.380,21.400,-41.368
C04828=1018.729,153.891,-135.741,-24.379,21.401,-41.372
C04829=1018.735,153.480,-135.700,-24.378,21.400,-41.375
C04830=1018.741,153.068,-135.661,-24.378,21.400,-41.377
C04831=1018.747,152.656,-135.621,-24.378,21.401,-41.381
C04832=1018.754,152.243,-135.581,-24.377,21.401,-41.383
C04833=1018.760,151.830,-135.540,-24.377,21.402,-41.387
C04834=1018.765,151.416,-135.501,-24.377,21.402,-41.389
C04835=1018.771,151.003,-135.461,-24.376,21.401,-41.392
C04836=1018.777,150.589,-135.420,-24.376,21.402,-41.394
C04837=1018.783,150.175,-135.380,-24.375,21.402,-41.398
C04838=1018.789,149.761,-135.340,-24.375,21.402,-41.401
C04839=1018.795,149.347,-135.300,-24.375,21.403,-41.403
C04840=1018.800,148.933,-135.260,-24.374,21.403,-41.407
C04841=1018.807,148.519,-135.220,-24.374,21.403,-41.409
C04842=1018.813,148.105,-135.180,-24.373,21.403,-41.412
C04843=1018.818,147.691,-135.139,-24.373,21.403,-41.416
C04844=1018.824,147.277,-135.099,-24.372,21.404,-41.418
C04845=1018.831,146.864,-135.059,-24.372,21.404,-41.422
C04846=1018.836,146.450,-135.019,-24.372,21.404,-41.424
C04847=1018.842,146.038,-134.978,-24.371,21.405,-41.427
C04848=1018.847,145.625,-134.938,-24.371,21.404,-41.431
C04849=1018.853,145.213,-134.899,-24.370,21.405,-41.432
C04850=1018.859,144.801,-134.859,-24.370,21.405,-41.436
C04851=1018.864,144.390,-134.820,-24.370,21.405,-41.438
C04852=1018.871,143.980,-134.780,-24.369,21.406,-41.442
C04853=1018.876,143.570,-134.740,-24.369,21.405,-41.445
C04854=1018.882,143.162,-134.700,-24.368,21.406,-41.448
C04855=1018.887,142.754,-134.661,-24.368,21.406,-41.451
C04856=1018.893,142.347,-134.621,-24.368,21.406,-41.453
C04857=1018.899,141.941,-134.582,-24.367,21.407,-41.457
C04858=1018.904,141.535,-134.543,-24.366,21.406,-41.460
C04859=1018.909,141.131,-134.504,-24.366,21.407,-41.462
C04860=1018.914,140.713,-134.463,-24.366,21.408,-41.466
C04861=1018.917,140.477,-134.441,-24.366,21.408,-41.468
C04862=1018.922,140.219,-134.415,-24.365,21.408,-41.470
C04863=1018.925,139.942,-134.389,-24.365,21.408,-41.471
C04864=1018.929,139.654,-134.361,-24.365,21.408,-41.473
C04865=1018.933,139.366,-134.334,-24.364,21.408,-41.475
C04866=1018.936,139.088,-134.306,-24.364,21.407,-41.476
C04867=1018.939,138.829,-134.281,-24.364,21.408,-41.478
C04868=1018.943,138.591,-134.259,-24.364,21.408,-41.480
C04869=1018.946,138.375,-134.238,-24.363,21.408,-41.482
C04870=1018.949,138.168,-134.218,-24.363,21.408,-41.484
C04871=1018.954,137.768,-134.179,-24.363,21.408,-41.486
C04872=1018.958,137.397,-134.143,-24.363,21.410,-41.488
C04873=1018.964,137.061,-134.111,-24.362,21.409,-41.491
C04874=1018.968,136.744,-134.081,-24.361,21.409,-41.495
C04875=1018.972,136.427,-134.049,-24.361,21.410,-41.497
C04876=1018.976,136.087,-134.017,-24.361,21.409,-41.500
C04877=1018.981,135.716,-133.981,-24.360,21.410,-41.502
C04878=1018.986,135.320,-133.943,-24.360,21.411,-41.505
C04879=1018.991,134.921,-133.904,-24.360,21.410,-41.508
C04880=1018.996,134.523,-133.866,-24.359,21.411,-41.510
C04881=1019.001,134.124,-133.828,-24.359,21.411,-41.514
C04882=1019.006,133.726,-133.790,-24.358,21.411,-41.517
C04883=1019.012,133.327,-133.751,-24.358,21.412,-41.519
C04884=1019.016,132.928,-133.713,-24.358,21.411,-41.523
C04885=1019.022,132.529,-133.674,-24.357,21.412,-41.525
C04886=1019.026,132.130,-133.636,-24.357,21.412,-41.528
C04887=1019.032,131.732,-133.597,-24.356,21.412,-41.532
C04888=1019.037,131.334,-133.559,-24.356,21.413,-41.534
C04889=1019.042,130.935,-133.521,-24.356,21.413,-41.538
C04890=1019.047,130.536,-133.482,-24.355,21.413,-41.541
C04891=1019.051,130.137,-133.444,-24.355,21.413,-41.543
C04892=1019.058,129.739,-133.406,-24.354,21.413,-41.547
C04893=1019.062,129.340,-133.368,-24.354,21.413,-41.550
C04894=1019.067,128.942,-133.329,-24.354,21.414,-41.552
C04895=1019.072,128.543,-133.290,-24.353,21.414,-41.555
C04896=1019.076,128.144,-133.252,-24.353,21.415,-41.558
C04897=1019.082,127.746,-133.215,-24.352,21.414,-41.561
C04898=1019.086,127.347,-133.176,-24.352,21.415,-41.565
C04899=1019.091,126.949,-133.138,-24.351,21.415,-41.567
C04900=1019.096,126.550,-133.099,-24.351,21.415,-41.571
C04901=1019.101,126.151,-133.061,-24.350,21.415,-41.574
C04902=1019.106,125.752,-133.023,-24.350,21.416,-41.576
C04903=1019.111,125.354,-132.985,-24.350,21.416,-41.580
C04904=1019.115,124.956,-132.947,-24.349,21.416,-41.583
C04905=1019.120,124.557,-132.909,-24.349,21.416,-41.585
C04906=1019.125,124.158,-132.870,-24.348,21.417,-41.589
C04907=1019.130,123.759,-132.832,-24.348,21.416,-41.592
C04908=1019.134,123.361,-132.793,-24.348,21.418,-41.595
C04909=1019.140,122.963,-132.756,-24.347,21.417,-41.598
C04910=1019.144,122.564,-132.717,-24.347,21.418,-41.602
C04911=1019.149,122.166,-132.679,-24.346,21.417,-41.605
C04912=1019.153,121.767,-132.641,-24.346,21.418,-41.607
C04913=1019.158,121.368,-132.602,-24.345,21.418,-41.611
C04914=1019.163,120.969,-132.565,-24.345,21.418,-41.614
C04915=1019.168,120.572,-132.527,-24.345,21.419,-41.617
C04916=1019.172,120.173,-132.488,-24.344,21.419,-41.620
C04917=1019.177,119.774,-132.451,-24.343,21.419,-41.624
C04918=1019.182,119.376,-132.413,-24.343,21.420,-41.626
C04919=1019.187,118.977,-132.375,-24.343,21.420,-41.629
C04920=1019.192,118.578,-132.337,-24.342,21.420,-41.633
C04921=1019.197,118.180,-132.299,-24.342,21.420,-41.637
C04922=1019.202,117.782,-132.261,-24.341,21.420,-41.638
C04923=1019.207,117.383,-132.224,-24.341,21.421,-41.642
C04924=1019.211,116.985,-132.186,-24.340,21.420,-41.646
C04925=1019.216,116.586,-132.148,-24.340,21.421,-41.649
C04926=1019.221,116.188,-132.110,-24.340,21.422,-41.652
C04927=1019.226,115.789,-132.073,-24.339,21.422,-41.655
C04928=1019.231,115.391,-132.035,-24.339,21.422,-41.659
C04929=1019.236,114.992,-131.997,-24.338,21.422,-41.662
C04930=1019.240,114.593,-131.959,-24.338,21.423,-41.664
C04931=1019.246,114.195,-131.921,-24.337,21.422,-41.668
C04932=1019.249,113.797,-131.883,-24.337,21.423,-41.671
C04933=1019.254,113.398,-131.846,-24.336,21.423,-41.675
C04934=1019.259,113.000,-131.808,-24.336,21.423,-41.677
C04935=1019.264,112.601,-131.770,-24.335,21.424,-41.681
C04936=1019.268,112.202,-131.732,-24.335,21.423,-41.684
C04937=1019.273,111.803,-131.695,-24.334,21.424,-41.688
C04938=1019.278,111.406,-131.657,-24.334,21.425,-41.690
C04939=1019.283,111.006,-131.619,-24.334,21.425,-41.694
C04940=1019.287,110.608,-131.582,-24.333,21.425,-41.697
C04941=1019.292,110.210,-131.544,-24.333,21.425,-41.701
C04942=1019.297,109.811,-131.506,-24.332,21.426,-41.703
C04943=1019.301,109.412,-131.469,-24.332,21.426,-41.707
C04944=1019.305,109.013,-131.431,-24.331,21.426,-41.710
C04945=1019.309,108.615,-131.393,-24.331,21.426,-41.714
C04946=1019.315,108.217,-131.356,-24.330,21.426,-41.717
C04947=1019.320,107.818,-131.318,-24.330,21.427,-41.719
C04948=1019.323,107.419,-131.280,-24.330,21.427,-41.723
C04949=1019.328,107.020,-131.243,-24.329,21.427,-41.727
C04950=1019.332,106.622,-131.205,-24.328,21.427,-41.730
C04951=1019.337,106.224,-131.168,-24.328,21.428,-41.734
C04952=1019.341,105.825,-131.131,-24.328,21.428,-41.736
C04953=1019.346,105.426,-131.092,-24.327,21.429,-41.740
C04954=1019.350,105.027,-131.055,-24.327,21.429,-41.743
C04955=1019.355,104.628,-131.017,-24.326,21.429,-41.747
C04956=1019.359,104.230,-130.980,-24.326,21.429,-41.751
C04957=1019.364,103.831,-130.942,-24.325,21.430,-41.754
C04958=1019.368,103.432,-130.905,-24.325,21.430,-41.756
C04959=1019.372,103.034,-130.867,-24.324,21.430,-41.760
C04960=1019.376,102.635,-130.830,-24.324,21.430,-41.763
C04961=1019.381,102.236,-130.792,-24.323,21.430,-41.767
C04962=1019.385,101.837,-130.754,-24.323,21.431,-41.771
C04963=1019.389,101.439,-130.717,-24.322,21.431,-41.775
C04964=1019.394,101.039,-130.679,-24.322,21.431,-41.778
C04965=1019.398,100.641,-130.642,-24.322,21.432,-41.780
C04966=1019.402,100.242,-130.605,-24.321,21.432,-41.784
C04967=1019.407,99.843,-130.567,-24.320,21.432,-41.787
C04968=1019.411,99.444,-130.530,-24.320,21.432,-41.791
C04969=1019.415,99.046,-130.493,-24.319,21.433,-41.795
C04970=1019.419,98.647,-130.454,-24.319,21.432,-41.798
C04971=1019.423,98.248,-130.417,-24.318,21.433,-41.802
C04972=1019.427,97.849,-130.380,-24.318,21.433,-41.806
C04973=1019.432,97.451,-130.343,-24.318,21.434,-41.808
C04974=1019.436,97.052,-130.306,-24.317,21.434,-41.811
C04975=1019.440,96.652,-130.268,-24.317,21.435,-41.815
C04976=1019.444,96.254,-130.230,-24.316,21.435,-41.819
C04977=1019.448,95.855,-130.193,-24.316,21.435,-41.822
C04978=1019.453,95.456,-130.156,-24.315,21.435,-41.826
C04979=1019.457,95.057,-130.119,-24.315,21.436,-41.830
C04980=1019.460,94.657,-130.081,-24.314,21.435,-41.833
C04981=1019.464,94.259,-130.044,-24.313,21.436,-41.837
C04982=1019.468,93.860,-130.007,-24.313,21.436,-41.841
C04983=1019.473,93.460,-129.969,-24.312,21.437,-41.844
C04984=1019.477,93.061,-129.932,-24.312,21.437,-41.846
C04985=1019.481,92.662,-129.895,-24.312,21.437,-41.850
C04986=1019.484,92.263,-129.857,-24.311,21.438,-41.854
C04987=1019.488,91.864,-129.820,-24.311,21.438,-41.857
C04988=1019.493,91.465,-129.783,-24.310,21.438,-41.861
C04989=1019.496,91.066,-129.746,-24.310,21.438,-41.865
C04990=1019.500,90.667,-129.709,-24.309,21.439,-41.868
C04991=1019.504,90.267,-129.671,-24.309,21.439,-41.872
C04992=1019.508,89.870,-129.634,-24.308,21.439,-41.875
C04993=1019.512,89.476,-129.597,-24.308,21.439,-41.879
C04994=1019.516,89.090,-129.562,-24.307,21.440,-41.883
C04995=1019.519,88.706,-129.526,-24.307,21.440,-41.887
C04996=1019.523,88.324,-129.490,-24.306,21.440,-41.890
C04997=1019.527,87.935,-129.454,-24.305,21.440,-41.894
C04998=1019.530,87.539,-129.417,-24.305,21.441,-41.898
C04999=1019.534,87.136,-129.379,-24.304,21.441,-41.901
C05000=1019.538,86.730,-129.342,-24.304,21.442,-41.905
C05001=1019.542,86.323,-129.304,-24.303,21.441,-41.908
C05002=1019.546,85.914,-129.265,-24.303,21.442,-41.912
C05003=1019.549,85.503,-129.228,-24.302,21.442,-41.916
C05004=1019.554,85.091,-129.190,-24.302,21.443,-41.920
C05005=1019.557,84.677,-129.151,-24.301,21.443,-41.923
C05006=1019.561,84.261,-129.113,-24.301,21.443,-41.927
C05007=1019.565,83.843,-129.073,-24.300,21.444,-41.931
C05008=1019.568,83.425,-129.035,-24.300,21.444,-41.935
C05009=1019.572,83.004,-128.996,-24.299,21.444,-41.938
C05010=1019.574,82.794,-128.976,-24.299,21.444,-41.940
C05011=1019.576,82.583,-128.957,-24.299,21.444,-41.942
C05012=1019.578,82.372,-128.937,-24.299,21.445,-41.944
C05013=1019.580,82.160,-128.917,-24.298,21.444,-41.947
C05014=1019.582,81.948,-128.898,-24.298,21.445,-41.949
C05015=1019.584,81.736,-128.878,-24.298,21.445,-41.951
C05016=1019.586,81.524,-128.858,-24.297,21.445,-41.953
C05017=1019.588,81.312,-128.839,-24.297,21.445,-41.955
C05018=1019.590,81.099,-128.820,-24.297,21.445,-41.956
C05019=1019.592,80.886,-128.799,-24.297,21.446,-41.958
C05020=1019.593,80.673,-128.780,-24.296,21.446,-41.960
C05021=1019.595,80.461,-128.760,-24.296,21.446,-41.962
C05022=1019.597,80.249,-128.740,-24.296,21.446,-41.964
C05023=1019.598,80.038,-128.721,-24.296,21.447,-41.966
C05024=1019.603,79.624,-128.683,-24.295,21.447,-41.970
C05025=1019.606,79.218,-128.645,-24.294,21.447,-41.973
C05026=1019.610,78.821,-128.608,-24.294,21.447,-41.977
C05027=1019.613,78.431,-128.573,-24.293,21.448,-41.980
C05028=1019.617,78.044,-128.537,-24.293,21.447,-41.986
C05029=1019.620,77.658,-128.502,-24.292,21.448,-41.989
C05030=1019.623,77.269,-128.465,-24.292,21.449,-41.994
C05031=1019.626,76.875,-128.429,-24.291,21.449,-41.997
C05032=1019.630,76.473,-128.392,-24.291,21.449,-42.001
C05033=1019.634,76.062,-128.354,-24.290,21.450,-42.004
C05034=1019.637,75.642,-128.315,-24.290,21.450,-42.008
C05035=1019.638,75.429,-128.296,-24.289,21.451,-42.010
C05036=1019.641,75.215,-128.276,-24.289,21.451,-42.012
C05037=1019.642,75.002,-128.256,-24.289,21.450,-42.015
C05038=1019.645,74.788,-128.237,-24.288,21.451,-42.017
C05039=1019.646,74.575,-128.217,-24.288,21.451,-42.019
C05040=1019.648,74.363,-128.198,-24.288,21.451,-42.021
C05041=1019.650,74.151,-128.178,-24.288,21.451,-42.023
C05042=1019.651,73.939,-128.159,-24.287,21.452,-42.025
C05043=1019.655,73.519,-128.120,-24.287,21.452,-42.028
C05044=1019.658,73.100,-128.082,-24.286,21.452,-42.034
C05045=1019.662,72.686,-128.043,-24.285,21.452,-42.037
C05046=1019.665,72.273,-128.005,-24.285,21.453,-42.041
C05047=1019.668,71.860,-127.967,-24.285,21.453,-42.045
C05048=1019.672,71.449,-127.930,-24.284,21.454,-42.049
C05049=1019.675,71.037,-127.892,-24.283,21.453,-42.054
C05050=1019.678,70.627,-127.854,-24.283,21.454,-42.058
C05051=1019.681,70.215,-127.816,-24.282,21.454,-42.061
C05052=1019.685,69.804,-127.779,-24.282,21.455,-42.065
C05053=1019.688,69.394,-127.741,-24.281,21.455,-42.069
C05054=1019.691,68.985,-127.703,-24.280,21.455,-42.074
C05055=1019.695,68.578,-127.666,-24.280,21.456,-42.078
C05056=1019.698,68.172,-127.629,-24.279,21.456,-42.082
C05057=1019.701,67.767,-127.592,-24.279,21.457,-42.085
C05058=1019.703,67.364,-127.555,-24.278,21.457,-42.089
C05059=1019.706,66.962,-127.518,-24.278,21.457,-42.094
C05060=1019.710,66.561,-127.482,-24.277,21.457,-42.098
C05061=1019.713,66.163,-127.445,-24.277,21.458,-42.102
C05062=1019.716,65.755,-127.408,-24.276,21.458,-42.106
C05063=1019.718,65.542,-127.389,-24.276,21.459,-42.108
C05064=1019.719,65.320,-127.369,-24.275,21.458,-42.111
C05065=1019.721,65.091,-127.348,-24.275,21.458,-42.113
C05066=1019.723,64.854,-127.326,-24.275,21.459,-42.115
C05067=1019.725,64.618,-127.304,-24.274,21.459,-42.116
C05068=1019.726,64.389,-127.283,-24.274,21.459,-42.120
C05069=1019.728,64.172,-127.264,-24.274,21.460,-42.122
C05070=1019.729,63.964,-127.245,-24.274,21.460,-42.124
C05071=1019.732,63.747,-127.225,-24.273,21.459,-42.127
C05072=1019.732,63.497,-127.203,-24.273,21.460,-42.129
C05073=1019.735,63.229,-127.178,-24.272,21.460,-42.131
C05074=1019.737,62.977,-127.155,-24.272,21.460,-42.133
C05075=1019.740,62.557,-127.117,-24.271,21.461,-42.139
C05076=1019.743,62.156,-127.080,-24.271,21.461,-42.142
C05077=1019.746,61.756,-127.044,-24.270,21.462,-42.146
C05078=1019.748,61.356,-127.007,-24.270,21.462,-42.150
C05079=1019.751,60.956,-126.971,-24.269,21.462,-42.155
C05080=1019.754,60.555,-126.935,-24.269,21.463,-42.159
C05081=1019.757,60.155,-126.899,-24.268,21.463,-42.163
C05082=1019.759,59.756,-126.862,-24.268,21.464,-42.166
C05083=1019.762,59.356,-126.825,-24.267,21.463,-42.172
C05084=1019.765,58.955,-126.789,-24.266,21.464,-42.175
C05085=1019.768,58.555,-126.753,-24.266,21.464,-42.179
C05086=1019.770,58.155,-126.716,-24.265,21.465,-42.183
C05087=1019.773,57.755,-126.680,-24.264,21.465,-42.188
C05088=1019.776,57.354,-126.644,-24.264,21.465,-42.192
C05089=1019.779,56.954,-126.608,-24.264,21.466,-42.196
C05090=1019.781,56.553,-126.572,-24.263,21.465,-42.201
C05091=1019.785,56.153,-126.536,-24.262,21.467,-42.205
C05092=1019.787,55.753,-126.499,-24.262,21.467,-42.209
C05093=1019.790,55.353,-126.463,-24.261,21.468,-42.212
C05094=1019.792,54.953,-126.427,-24.260,21.468,-42.218
C05095=1019.795,54.553,-126.391,-24.260,21.468,-42.221
C05096=1019.797,54.152,-126.355,-24.259,21.468,-42.225
C05097=1019.800,53.753,-126.318,-24.259,21.468,-42.230
C05098=1019.803,53.352,-126.282,-24.258,21.469,-42.234
C05099=1019.805,52.952,-126.246,-24.258,21.469,-42.238
C05100=1019.808,52.552,-126.210,-24.257,21.469,-42.243
C05101=1019.811,52.152,-126.174,-24.256,21.470,-42.247
C05102=1019.812,51.752,-126.138,-24.256,21.471,-42.251
C05103=1019.816,51.352,-126.102,-24.255,21.471,-42.255
C05104=1019.818,50.951,-126.065,-24.255,21.471,-42.260
C05105=1019.820,50.551,-126.030,-24.254,21.472,-42.264
C05106=1019.823,50.151,-125.994,-24.254,21.472,-42.268
C05107=1019.825,49.750,-125.958,-24.253,21.472,-42.273
C05108=1019.828,49.351,-125.922,-24.252,21.473,-42.277
C05109=1019.830,48.950,-125.886,-24.251,21.472,-42.282
C05110=1019.833,48.551,-125.850,-24.251,21.474,-42.286
C05111=1019.834,48.150,-125.814,-24.251,21.474,-42.290
C05112=1019.837,47.750,-125.778,-24.250,21.474,-42.295
C05113=1019.839,47.350,-125.743,-24.249,21.475,-42.299
C05114=1019.843,46.950,-125.707,-24.249,21.475,-42.302
C05115=1019.844,46.549,-125.671,-24.248,21.475,-42.308
C05116=1019.847,46.150,-125.635,-24.247,21.475,-42.311
C05117=1019.849,45.749,-125.599,-24.247,21.477,-42.316
C05118=1019.851,45.350,-125.563,-24.246,21.477,-42.321
C05119=1019.853,44.950,-125.527,-24.246,21.477,-42.325
C05120=1019.855,44.550,-125.492,-24.245,21.477,-42.330
C05121=1019.858,44.149,-125.456,-24.244,21.477,-42.333
C05122=1019.861,43.749,-125.421,-24.244,21.479,-42.338
C05123=1019.862,43.349,-125.385,-24.243,21.479,-42.343
C05124=1019.865,42.950,-125.349,-24.243,21.479,-42.347
C05125=1019.866,42.549,-125.313,-24.242,21.479,-42.352
C05126=1019.869,42.149,-125.277,-24.241,21.479,-42.356
C05127=1019.871,41.749,-125.241,-24.241,21.480,-42.359
C05128=1019.874,41.349,-125.206,-24.240,21.481,-42.365
C05129=1019.875,40.949,-125.171,-24.240,21.481,-42.369
C05130=1019.878,40.549,-125.135,-24.239,21.481,-42.374
C05131=1019.880,40.150,-125.100,-24.238,21.481,-42.378
C05132=1019.882,39.750,-125.064,-24.238,21.482,-42.383
C05133=1019.884,39.350,-125.028,-24.237,21.483,-42.387
C05134=1019.886,38.950,-124.992,-24.237,21.483,-42.391
C05135=1019.888,38.550,-124.958,-24.236,21.483,-42.396
C05136=1019.890,38.150,-124.922,-24.235,21.483,-42.400
C05137=1019.892,37.750,-124.887,-24.235,21.484,-42.405
C05138=1019.894,37.351,-124.851,-24.234,21.485,-42.409
C05139=1019.896,36.950,-124.815,-24.233,21.484,-42.414
C05140=1019.898,36.551,-124.780,-24.233,21.485,-42.418
C05141=1019.899,36.151,-124.744,-24.232,21.486,-42.424
C05142=1019.902,35.751,-124.710,-24.231,21.486,-42.428
C05143=1019.904,35.351,-124.674,-24.231,21.486,-42.433
C05144=1019.905,34.951,-124.639,-24.230,21.486,-42.437
C05145=1019.908,34.552,-124.603,-24.229,21.487,-42.442
C05146=1019.910,34.152,-124.568,-24.229,21.488,-42.446
C05147=1019.911,33.752,-124.532,-24.228,21.487,-42.451
C05148=1019.913,33.353,-124.497,-24.228,21.489,-42.455
C05149=1019.915,32.953,-124.463,-24.227,21.489,-42.461
C05150=1019.917,32.553,-124.427,-24.226,21.489,-42.464
C05151=1019.918,32.153,-124.392,-24.226,21.489,-42.469
C05152=1019.921,31.754,-124.356,-24.225,21.490,-42.474
C05153=1019.922,31.355,-124.321,-24.224,21.490,-42.479
C05154=1019.923,30.955,-124.286,-24.224,21.491,-42.483
C05155=1019.926,30.555,-124.251,-24.223,21.491,-42.488
C05156=1019.927,30.156,-124.216,-24.223,21.492,-42.492
C05157=1019.929,29.756,-124.181,-24.222,21.492,-42.497
C05158=1019.931,29.356,-124.145,-24.221,21.492,-42.501
C05159=1019.931,29.256,-124.137,-24.221,21.492,-42.503
C05160=1020.012,-28.690,-119.243,-24.120,21.563,-43.247
C05161=1020.012,-29.013,-119.217,-24.119,21.563,-43.250
C05162=1020.011,-29.335,-119.190,-24.119,21.565,-43.255
C05163=1020.010,-29.733,-119.158,-24.118,21.565,-43.260
C05164=1020.009,-30.130,-119.126,-24.117,21.565,-43.265
C05165=1020.009,-30.528,-119.094,-24.117,21.566,-43.271
C05166=1020.008,-30.925,-119.062,-24.116,21.567,-43.277
C05167=1020.007,-31.322,-119.030,-24.115,21.568,-43.282
C05168=1020.007,-31.720,-118.998,-24.114,21.567,-43.287
C05169=1020.006,-32.117,-118.966,-24.114,21.568,-43.293
C05170=1020.005,-32.515,-118.934,-24.113,21.569,-43.299
C05171=1020.004,-32.912,-118.902,-24.112,21.570,-43.304
C05172=1020.004,-33.310,-118.870,-24.111,21.570,-43.310
C05173=1020.003,-33.707,-118.838,-24.111,21.570,-43.315
C05174=1020.001,-34.104,-118.806,-24.110,21.571,-43.321
C05175=1020.001,-34.501,-118.774,-24.109,21.571,-43.328
C05176=1020.000,-34.899,-118.743,-24.108,21.572,-43.334
C05177=1019.999,-35.296,-118.711,-24.107,21.572,-43.339
C05178=1019.998,-35.693,-118.679,-24.107,21.573,-43.344
C05179=1019.997,-36.091,-118.648,-24.106,21.573,-43.350
C05180=1019.997,-36.488,-118.615,-24.105,21.574,-43.356
C05181=1019.995,-36.885,-118.584,-24.105,21.575,-43.361
C05182=1019.995,-37.283,-118.552,-24.104,21.575,-43.366
C05183=1019.993,-37.680,-118.521,-24.103,21.576,-43.372
C05184=1019.992,-38.078,-118.488,-24.102,21.576,-43.378
C05185=1019.990,-38.475,-118.457,-24.102,21.577,-43.383
C05186=1019.990,-38.873,-118.425,-24.101,21.578,-43.389
C05187=1019.988,-39.270,-118.393,-24.100,21.578,-43.394
C05188=1019.988,-39.667,-118.362,-24.099,21.579,-43.400
C05189=1019.986,-40.064,-118.330,-24.099,21.579,-43.405
C05190=1019.985,-40.461,-118.299,-24.098,21.580,-43.411
C05191=1019.984,-40.859,-118.267,-24.097,21.581,-43.417
C05192=1019.983,-41.256,-118.236,-24.096,21.582,-43.422
C05193=1019.981,-41.653,-118.204,-24.096,21.582,-43.427
C05194=1019.981,-42.051,-118.173,-24.095,21.582,-43.433
C05195=1019.979,-42.448,-118.141,-24.094,21.583,-43.439
C05196=1019.978,-42.845,-118.110,-24.093,21.584,-43.444
C05197=1019.977,-43.242,-118.079,-24.092,21.584,-43.451
C05198=1019.975,-43.639,-118.047,-24.092,21.585,-43.457
C05199=1019.974,-44.037,-118.016,-24.091,21.585,-43.462
C05200=1019.973,-44.434,-117.985,-24.090,21.585,-43.468
C05201=1019.971,-44.831,-117.953,-24.089,21.586,-43.473
C05202=1019.970,-45.228,-117.922,-24.089,21.587,-43.479
C05203=1019.968,-45.625,-117.891,-24.088,21.588,-43.485
C05204=1019.967,-46.023,-117.860,-24.087,21.589,-43.490
C05205=1019.966,-46.420,-117.828,-24.086,21.588,-43.496
C05206=1019.964,-46.817,-117.797,-24.086,21.589,-43.501
C05207=1019.963,-47.214,-117.766,-24.085,21.590,-43.507
C05208=1019.961,-47.611,-117.734,-24.084,21.591,-43.512
C05209=1019.960,-48.009,-117.703,-24.084,21.592,-43.518
C05210=1019.958,-48.404,-117.673,-24.083,21.592,-43.525
C05211=1019.957,-48.802,-117.642,-24.082,21.592,-43.531
C05212=1019.956,-49.199,-117.610,-24.081,21.592,-43.536
C05213=1019.955,-49.596,-117.579,-24.080,21.593,-43.542
C05214=1019.952,-49.993,-117.548,-24.080,21.594,-43.547
C05215=1019.951,-50.390,-117.517,-24.079,21.595,-43.553
C05216=1019.949,-50.787,-117.486,-24.078,21.595,-43.558
C05217=1019.947,-51.184,-117.455,-24.077,21.596,-43.564
C05218=1019.946,-51.582,-117.424,-24.077,21.597,-43.570
C05219=1019.944,-51.978,-117.393,-24.076,21.598,-43.575
C05220=1019.942,-52.374,-117.362,-24.075,21.598,-43.581
C05221=1019.941,-52.772,-117.331,-24.074,21.598,-43.588
C05222=1019.939,-53.168,-117.300,-24.073,21.599,-43.593
C05223=1019.938,-53.566,-117.270,-24.073,21.599,-43.599
C05224=1019.935,-53.963,-117.239,-24.072,21.600,-43.604
C05225=1019.933,-54.360,-117.208,-24.071,21.601,-43.610
C05226=1019.932,-54.757,-117.177,-24.071,21.602,-43.616
C05227=1019.930,-55.154,-117.146,-24.070,21.603,-43.621
C05228=1019.928,-55.551,-117.115,-24.069,21.602,-43.627
C05229=1019.927,-55.948,-117.085,-24.068,21.603,-43.632
C05230=1019.924,-56.346,-117.054,-24.067,21.603,-43.639
C05231=1019.923,-56.744,-117.023,-24.067,21.604,-43.645
C05232=1019.921,-57.142,-116.993,-24.066,21.605,-43.651
C05233=1019.918,-57.541,-116.961,-24.065,21.606,-43.656
C05234=1019.917,-57.940,-116.931,-24.064,21.606,-43.662
C05235=1019.915,-58.340,-116.900,-24.064,21.607,-43.667
C05236=1019.912,-58.741,-116.869,-24.063,21.608,-43.673
C05237=1019.911,-59.141,-116.838,-24.062,21.608,-43.680
C05238=1019.908,-59.542,-116.807,-24.061,21.609,-43.686
C05239=1019.907,-59.944,-116.777,-24.061,21.610,-43.691
C05240=1019.904,-60.346,-116.745,-24.060,21.610,-43.697
C05241=1019.902,-60.750,-116.715,-24.059,21.610,-43.702
C05242=1019.899,-61.153,-116.684,-24.058,21.611,-43.708
C05243=1019.897,-61.557,-116.653,-24.057,21.611,-43.715
C05244=1019.895,-61.962,-116.622,-24.057,21.612,-43.720
C05245=1019.893,-62.367,-116.590,-24.056,21.613,-43.726
C05246=1019.891,-62.773,-116.560,-24.055,21.614,-43.732
C05247=1019.889,-63.179,-116.529,-24.054,21.615,-43.737
C05248=1019.887,-63.585,-116.498,-24.053,21.615,-43.744
C05249=1019.884,-63.993,-116.467,-24.053,21.615,-43.750
C05250=1019.882,-64.400,-116.435,-24.052,21.616,-43.756
C05251=1019.879,-64.808,-116.404,-24.051,21.617,-43.761
C05252=1019.877,-65.217,-116.373,-24.050,21.617,-43.768
C05253=1019.874,-65.626,-116.341,-24.049,21.618,-43.774
C05254=1019.872,-66.035,-116.311,-24.049,21.619,-43.780
C05255=1019.870,-66.445,-116.280,-24.048,21.620,-43.785
C05256=1019.867,-66.855,-116.248,-24.047,21.620,-43.791
C05257=1019.865,-67.264,-116.217,-24.046,21.621,-43.798
C05258=1019.862,-67.674,-116.186,-24.046,21.621,-43.804
C05259=1019.859,-68.085,-116.155,-24.045,21.622,-43.809
C05260=1019.856,-68.495,-116.124,-24.044,21.623,-43.815
C05261=1019.854,-68.906,-116.093,-24.043,21.623,-43.822
C05262=1019.851,-69.316,-116.061,-24.042,21.624,-43.827
C05263=1019.848,-69.728,-116.030,-24.042,21.625,-43.833
C05264=1019.846,-70.138,-116.000,-24.041,21.625,-43.839
C05265=1019.843,-70.550,-115.968,-24.040,21.626,-43.846
C05266=1019.841,-70.961,-115.937,-24.039,21.626,-43.851
C05267=1019.837,-71.371,-115.906,-24.039,21.627,-43.857
C05268=1019.835,-71.782,-115.875,-24.038,21.628,-43.865
C05269=1019.832,-72.193,-115.844,-24.037,21.629,-43.870
C05270=1019.829,-72.604,-115.814,-24.036,21.630,-43.876
C05271=1019.827,-73.014,-115.783,-24.035,21.631,-43.881
C05272=1019.823,-73.425,-115.751,-24.034,21.631,-43.888
C05273=1019.821,-73.836,-115.721,-24.034,21.632,-43.894
C05274=1019.818,-74.246,-115.690,-24.033,21.632,-43.900
C05275=1019.815,-74.656,-115.659,-24.032,21.633,-43.905
C05276=1019.812,-75.066,-115.628,-24.031,21.633,-43.912
C05277=1019.809,-75.477,-115.598,-24.031,21.634,-43.918
C05278=1019.806,-75.886,-115.567,-24.030,21.635,-43.924
C05279=1019.803,-76.295,-115.536,-24.029,21.636,-43.929
C05280=1019.800,-76.704,-115.506,-24.028,21.636,-43.936
C05281=1019.797,-77.113,-115.475,-24.027,21.637,-43.942
C05282=1019.794,-77.521,-115.445,-24.027,21.637,-43.948
C05283=1019.790,-77.929,-115.414,-24.026,21.638,-43.953
C05284=1019.788,-78.337,-115.384,-24.025,21.638,-43.960
C05285=1019.784,-78.744,-115.354,-24.024,21.639,-43.966
C05286=1019.781,-79.150,-115.323,-24.023,21.640,-43.972
C05287=1019.778,-79.557,-115.293,-24.023,21.641,-43.977
C05288=1019.775,-79.963,-115.263,-24.022,21.641,-43.984
C05289=1019.772,-80.367,-115.233,-24.021,21.642,-43.990
C05290=1019.768,-80.771,-115.203,-24.020,21.643,-43.995
C05291=1019.765,-81.175,-115.173,-24.020,21.643,-44.001
C05292=1019.762,-81.579,-115.143,-24.019,21.644,-44.007
C05293=1019.758,-81.981,-115.113,-24.018,21.644,-44.014
C05294=1019.755,-82.384,-115.083,-24.017,21.645,-44.019
C05295=1019.752,-82.786,-115.053,-24.016,21.646,-44.025
C05296=1019.748,-83.186,-115.024,-24.016,21.647,-44.031
C05297=1019.745,-83.586,-114.994,-24.015,21.648,-44.036
C05298=1019.742,-83.986,-114.965,-24.014,21.648,-44.043
C05299=1019.739,-84.392,-114.934,-24.013,21.649,-44.049
C05300=1019.737,-84.615,-114.918,-24.013,21.649,-44.053
C05301=1019.734,-84.857,-114.900,-24.012,21.650,-44.056
C05302=1019.732,-85.110,-114.882,-24.012,21.649,-44.060
C05303=1019.730,-85.365,-114.863,-24.012,21.650,-44.062
C05304=1019.728,-85.611,-114.845,-24.011,21.650,-44.065
C05305=1019.726,-85.841,-114.827,-24.011,21.651,-44.069
C05306=1019.723,-86.250,-114.798,-24.010,21.652,-44.077
C05307=1019.719,-86.638,-114.769,-24.009,21.652,-44.082
C05308=1019.716,-87.017,-114.741,-24.008,21.652,-44.087
C05309=1019.712,-87.391,-114.714,-24.007,21.653,-44.093
C05310=1019.709,-87.762,-114.687,-24.007,21.654,-44.099
C05311=1019.706,-88.137,-114.659,-24.006,21.655,-44.104
C05312=1019.703,-88.544,-114.629,-24.005,21.656,-44.112
C05313=1019.700,-88.793,-114.611,-24.005,21.656,-44.116
C05314=1019.697,-89.067,-114.591,-24.004,21.657,-44.117
C05315=1019.695,-89.350,-114.570,-24.004,21.656,-44.121
C05316=1019.692,-89.626,-114.550,-24.003,21.657,-44.124
C05317=1019.690,-89.876,-114.532,-24.003,21.657,-44.128
C05318=1019.688,-90.095,-114.516,-24.002,21.658,-44.132
C05319=1019.684,-90.490,-114.487,-24.002,21.659,-44.138
C05320=1019.680,-90.884,-114.458,-24.001,21.659,-44.145
C05321=1019.676,-91.276,-114.429,-24.000,21.660,-44.150
C05322=1019.673,-91.668,-114.401,-23.999,21.660,-44.156
C05323=1019.669,-92.060,-114.372,-23.999,21.661,-44.162
C05324=1019.666,-92.451,-114.344,-23.998,21.662,-44.167
C05325=1019.661,-92.841,-114.315,-23.997,21.663,-44.173
C05326=1019.658,-93.230,-114.287,-23.996,21.664,-44.178
C05327=1019.654,-93.618,-114.259,-23.996,21.664,-44.184
C05328=1019.650,-94.006,-114.230,-23.995,21.664,-44.189
C05329=1019.646,-94.393,-114.202,-23.994,21.665,-44.195
C05330=1019.642,-94.778,-114.175,-23.994,21.666,-44.200
C05331=1019.639,-95.164,-114.147,-23.993,21.666,-44.207
C05332=1019.634,-95.549,-114.118,-23.992,21.667,-44.213
C05333=1019.630,-95.934,-114.090,-23.991,21.668,-44.219
C05334=1019.626,-96.318,-114.063,-23.990,21.668,-44.224
C05335=1019.623,-96.701,-114.035,-23.990,21.669,-44.230
C05336=1019.618,-97.085,-114.007,-23.989,21.669,-44.235
C05337=1019.615,-97.468,-113.980,-23.988,21.670,-44.241
C05338=1019.611,-97.852,-113.951,-23.988,21.671,-44.246
C05339=1019.607,-98.235,-113.924,-23.987,21.672,-44.252
C05340=1019.602,-98.617,-113.897,-23.986,21.673,-44.258
C05341=1019.599,-99.002,-113.869,-23.985,21.673,-44.263
C05342=1019.594,-99.385,-113.840,-23.985,21.673,-44.268
C05343=1019.590,-99.769,-113.813,-23.984,21.674,-44.274
C05344=1019.586,-100.154,-113.786,-23.983,21.675,-44.280
C05345=1019.582,-100.539,-113.758,-23.982,21.676,-44.285
C05346=1019.578,-100.925,-113.730,-23.982,21.677,-44.291
C05347=1019.574,-101.310,-113.702,-23.981,21.676,-44.296
C05348=1019.569,-101.698,-113.675,-23.980,21.677,-44.302
C05349=1019.565,-102.086,-113.647,-23.980,21.678,-44.307
C05350=1019.560,-102.474,-113.619,-23.979,21.678,-44.314
C05351=1019.556,-102.863,-113.591,-23.978,21.679,-44.320
C05352=1019.552,-103.253,-113.563,-23.977,21.680,-44.326
C05353=1019.547,-103.643,-113.535,-23.976,21.681,-44.331
C05354=1019.543,-104.034,-113.507,-23.976,21.682,-44.337
C05355=1019.538,-104.426,-113.479,-23.975,21.681,-44.342
C05356=1019.534,-104.818,-113.451,-23.974,21.682,-44.348
C05357=1019.529,-105.211,-113.424,-23.974,21.683,-44.353
C05358=1019.525,-105.603,-113.396,-23.973,21.684,-44.359
C05359=1019.520,-105.996,-113.367,-23.972,21.685,-44.365
C05360=1019.515,-106.389,-113.339,-23.971,21.686,-44.370
C05361=1019.511,-106.781,-113.312,-23.971,21.686,-44.376
C05362=1019.507,-107.175,-113.283,-23.970,21.687,-44.383
C05363=1019.502,-107.568,-113.255,-23.969,21.687,-44.388
C05364=1019.496,-107.961,-113.227,-23.968,21.688,-44.394
C05365=1019.492,-108.353,-113.200,-23.968,21.688,-44.399
C05366=1019.487,-108.746,-113.172,-23.967,21.689,-44.405
C05367=1019.482,-109.139,-113.144,-23.966,21.690,-44.411
C05368=1019.477,-109.531,-113.116,-23.965,21.691,-44.416
C05369=1019.472,-109.924,-113.088,-23.965,21.691,-44.422
